discrete alarms
   1: '1000 Betriebsfehler liegt vor / 1000 Operation Error / 1000 Erreur de fonctionnement', class Errors, trigger "WP231PR_DB_s_IO_DATA_OPERATION_ERRORS" bit 0
   2: 'Betriebsfehler Byte 1 Bit 1 / Operation Error Byte 1 Bit 1 / 1101 Court circuit pesons', class Errors, trigger "WP231PR_DB_s_IO_DATA_OPERATION_ERRORS" bit 1
   3: '1104 ADC Sense-Spannung zu gering / 1104 ADC sense voltage too low / 1104 Tension capteurs CAN trop basse', class Errors, trigger "WP231PR_DB_s_IO_DATA_OPERATION_ERRORS" bit 2
   4: 'Betriebsfehler Byte 1 Bit 3 / Operation Error Byte 1 Bit 1 / 1101 Court circuit pesons', class Errors, trigger "WP231PR_DB_s_IO_DATA_OPERATION_ERRORS" bit 3
   5: '1105 ADC Ausserhalb zulässigem Digit-Bereich (positiv) / 1105 ADC out of range (positive) / 1105 CAN hors plage de mesure (max)', class Errors, trigger "WP231PR_DB_s_IO_DATA_OPERATION_ERRORS" bit 4
   6: '1106 ADC Ausserhalb zulässigem Digit-Bereich (negativ) / 1106 ADC out of range (negative) / 1106 CAN hors plage de mesure (min)', class Errors, trigger "WP231PR_DB_s_IO_DATA_OPERATION_ERRORS" bit 5
   7: '1002 RAM-Fehler / 1002 RAM error / 1002 Erreur RAM', class Errors, trigger "WP231PR_DB_s_IO_DATA_OPERATION_ERRORS" bit 6
   8: '1102 ADC Fehler / 1102 ADC error / 1102 Erreur CAN', class Errors, trigger "WP231PR_DB_s_IO_DATA_OPERATION_ERRORS" bit 7
   9: '1005 Prozessalarm verloren / 1005 Processalarm lost / 1005 Perte des messages processus', class Errors, trigger "WP231PR_DB_s_IO_DATA_OPERATION_ERRORS" bit 8
   10: '1003 Checksummenfehler Daten / 1003 Checksum error data / 1003 Erreur données checksum', class Errors, trigger "WP231PR_DB_s_IO_DATA_OPERATION_ERRORS" bit 9
   11: '1107 Eichfähige HMI-Anzeige ist ausgefallen / 1107 Legal-for-trade display disturbed / 1107 Perte de l'affichage légal sur le pupitre HMI', class Errors, trigger "WP231PR_DB_s_IO_DATA_OPERATION_ERRORS" bit 10
   12: '1004 Checksummenfehler Programm / 1004 Checksum error program / 1004 Erreur données checksum du programme', class Errors, trigger "WP231PR_DB_s_IO_DATA_OPERATION_ERRORS" bit 11
   13: '1006 Fehler Logbuch / 1006 Error log-book / 1006 Erreur sur le cahier des rapports', class Errors, trigger "WP231PR_DB_s_IO_DATA_OPERATION_ERRORS" bit 12
   14: '1001 Reset nach Fehler (Watchdog Error) / 1001 Restart after failure (watchdog error) / 1001 Reset après erreur (Watchdog)', class Errors, trigger "WP231PR_DB_s_IO_DATA_OPERATION_ERRORS" bit 13
   15: '1007 Falsche Applikations-ID / 1007 Wrong application ID / 1007 Erreur ID de l'application', class Errors, trigger "WP231PR_DB_s_IO_DATA_OPERATION_ERRORS" bit 14
   16: 'Betriebsfehlerbyte 2 Bit 7 / Operation Error Byte 2 Bit 7 / Erreur fonctionnement octet 2 bit 7', class Errors, trigger "WP231PR_DB_s_IO_DATA_OPERATION_ERRORS" bit 15
   17: '2000 Technologiefehler / 2000 Technological error / 2000 Erreur technologique', class Errors, trigger "WP231PR_DB_s_IO_DATA_TECHNOLOGICAL_ERRORS" bit 0
   18: '2001 Timeout Tarieren oder Nullstellen / 2001 Timeout tare or zero setting / 2001 Timeout tarage ou RAZ (temps d'attente dépassé)', class Errors, trigger "WP231PR_DB_s_IO_DATA_TECHNOLOGICAL_ERRORS" bit 1
   19: '2002 Trace überlastet / 2002 Trace overloaded / 2002 Mémoire trace pleine', class Errors, trigger "WP231PR_DB_s_IO_DATA_TECHNOLOGICAL_ERRORS" bit 2
   20: '2003 Einschaltnullsetzen nicht möglich / 2003 Initial Zeroing not possible / 2003 RAZ à la mise sous tension impossible', class Errors, trigger "WP231PR_DB_s_IO_DATA_TECHNOLOGICAL_ERRORS" bit 3
   21: 'Technologiefehlerbyte 1 Bit 4 / Technological error Byte 1 Bit 4 / Erreur technologique octet 1 bit 4', class Errors, trigger "WP231PR_DB_s_IO_DATA_TECHNOLOGICAL_ERRORS" bit 4
   22: 'Technologiefehlerbyte 1 Bit 5 / Technological error Byte 1 Bit 5 / Erreur technologique octet 1 bit 5', class Errors, trigger "WP231PR_DB_s_IO_DATA_TECHNOLOGICAL_ERRORS" bit 5
   23: 'Technologiefehlerbyte 1 Bit 6 / Technological error Byte 1 Bit 6 / Erreur technologique octet 1 bit 6', class Errors, trigger "WP231PR_DB_s_IO_DATA_TECHNOLOGICAL_ERRORS" bit 6
   24: 'Technologiefehlerbyte 1 Bit 7 / Technological error Byte 1 Bit 7 / Erreur technologique octet 1 bit 7', class Errors, trigger "WP231PR_DB_s_IO_DATA_TECHNOLOGICAL_ERRORS" bit 7
   25: 'Technologiefehlerbyte 1 Bit 7 / Technological error Byte 2 Bit 0 / Erreur technologique octet 2 bit 0', class Errors, trigger "WP231PR_DB_s_IO_DATA_TECHNOLOGICAL_ERRORS" bit 8
   26: 'Technologiefehlerbyte 2 Bit 1 / Technological error Byte 2 Bit 1 / Erreur technologique octet 2 bit 1', class Errors, trigger "WP231PR_DB_s_IO_DATA_TECHNOLOGICAL_ERRORS" bit 9
   27: 'Technologiefehlerbyte 2 Bit 2 / Technological error Byte 2 Bit 2 / Erreur technologique octet 2 bit 2', class Errors, trigger "WP231PR_DB_s_IO_DATA_TECHNOLOGICAL_ERRORS" bit 10
   28: 'Technologiefehlerbyte 2 Bit 3 / Technological error Byte 2 Bit 3 / Erreur technologique octet 2 bit 3', class Errors, trigger "WP231PR_DB_s_IO_DATA_TECHNOLOGICAL_ERRORS" bit 11
   29: 'Technologiefehlerbyte 2 Bit 4 / Technological error Byte 2 Bit 4 / Erreur technologique octet 2 bit 4', class Errors, trigger "WP231PR_DB_s_IO_DATA_TECHNOLOGICAL_ERRORS" bit 12
   30: 'Technologiefehlerbyte 2 Bit 5 / Technological error Byte 2 Bit 5 / Erreur technologique octet 2 bit 5', class Errors, trigger "WP231PR_DB_s_IO_DATA_TECHNOLOGICAL_ERRORS" bit 13
   31: 'Technologiefehlerbyte 2 Bit 6 / Technological error Byte 2 Bit 6 / Erreur technologique octet 2 bit 6', class Errors, trigger "WP231PR_DB_s_IO_DATA_TECHNOLOGICAL_ERRORS" bit 14
   32: 'Technologiefehlerbyte 2 Bit 7 / Technological error Byte 2 Bit 7 / Erreur technologique octet 2 bit 7', class Errors, trigger "WP231PR_DB_s_IO_DATA_TECHNOLOGICAL_ERRORS" bit 15
   33: '5000 Daten- oder Bedienfehler / 5000 Data or command error / 5000 Erreur données ou utilisateur', class Errors, trigger "WP231PR_DB_s_IO_DATA_DATA_CMD_ERROR_1" bit 0
   34: '5001 Befehlscode oder Datensatz nicht bekannt / 5001 Data record or command unknown / 5001 Ordre ou numéro de DR inconnu', class Errors, trigger "WP231PR_DB_s_IO_DATA_DATA_CMD_ERROR_1" bit 1
   35: '5002 Befehl oder Datenänderung nicht erlaubt, da Schreibschutz aktiv / 5002 Command or Data modification not allowed / 5002 Ordre ou modification des paramètres interdit parce que la protection en écriture est activée', class Errors, trigger "WP231PR_DB_s_IO_DATA_DATA_CMD_ERROR_1" bit 2
   36: '5003 Verlassen des Servicebetriebs unzulässig, da Justage nicht abgeschlossen / 5003 Service Mode can't be switched off, as calibration was not completed / 5003 Impossible de quitter le mode service parce que l'étalonnage n'est pas terminé', class Errors, trigger "WP231PR_DB_s_IO_DATA_DATA_CMD_ERROR_1" bit 3
   37: '5004 Befehl oder Datenübertragung nur im Servicebetrieb möglich / 5004 Command or data transfer only permitted in service mode / 5004 Ordre ou transmission de données uniquement possible en mode service', class Errors, trigger "WP231PR_DB_s_IO_DATA_DATA_CMD_ERROR_1" bit 4
   38: '5005 Befehl oder Datenübertragung im Servicebetrieb nicht möglich, da Servicebetrieb aktiv / 5005 Command or data transfer not permitted in service mode / 5005 Ordre ou transmission de données impossible parce que le mode service est activé', class Errors, trigger "WP231PR_DB_s_IO_DATA_DATA_CMD_ERROR_1" bit 5
   39: '5006 Befehl oder Datenübertragung nicht möglich da BUSY / 5006 Command or data transfer not possible while BUSY / 5006 Ordre ou transmission de données impossible parce que la CPU est en mode stop ou erreur', class Errors, trigger "WP231PR_DB_s_IO_DATA_DATA_CMD_ERROR_1" bit 6
   40: '5007 Befehl oder Datenübertragung nicht möglich da Modul gestört oder CPU in Stop / 5007 Command or data transfer not possible because of error or CPU stop / 5007 Ordre ou transmission de données impossible parce que le module est en mode BUSY', class Errors, trigger "WP231PR_DB_s_IO_DATA_DATA_CMD_ERROR_1" bit 7
   41: 'Daten-Bedienfehler Byte 2 Bit 0 / Data Command Error Byte 2 Bit 0 / Erreur de données/d'utilisation octet 2 bit 0', class Errors, trigger "WP231PR_DB_s_IO_DATA_DATA_CMD_ERROR_1" bit 8
   42: '5103 Befehl nicht möglich, da Eichanzeige fehlt oder nicht sichtbar / 5103 Command not possible - SecureDisplay is missing or hidden / 5103 Ordre impossible parce que l'afficheur légal manque ou n'est pas disponible', class Errors, trigger "WP231PR_DB_s_IO_DATA_DATA_CMD_ERROR_1" bit 9
   43: '5101 Befehle in diesem Zustand nicht möglich / 5101 Command in this state not possible / 5101 Ordre impossible dans cet état', class Errors, trigger "WP231PR_DB_s_IO_DATA_DATA_CMD_ERROR_1" bit 10
   44: '5102 Befehl nicht möglich, da kein Stillstand vorliegt / 5102 Command not possible - No Standstill / 5102 Ordre impossible parce que l'état stable n'est pas atteint', class Errors, trigger "WP231PR_DB_s_IO_DATA_DATA_CMD_ERROR_1" bit 11
   45: '5104 Befehl nicht möglich, da Bereich überschritten / 5104 Command not possible - Limit exceeded / 5104 Ordre impossible parce que la plage de mesure est dépassée', class Errors, trigger "WP231PR_DB_s_IO_DATA_DATA_CMD_ERROR_1" bit 12
   46: '5105 Wägezellenparameter nicht plausibel / 5105 Load cell parameter not plausible / 5105 Les paramètres pesons ne sont pas plausibles', class Errors, trigger "WP231PR_DB_s_IO_DATA_DATA_CMD_ERROR_1" bit 13
   47: 'Daten-Bedienfehler Byte 2 Bit 0 / Data Command Error Byte 2 Bit 6 / Erreur de données/d'utilisation octet 2 bit 6', class Errors, trigger "WP231PR_DB_s_IO_DATA_DATA_CMD_ERROR_1" bit 14
   48: '5107 Kennlinienverschiebung nicht möglich / 5107 Calibration charcteristic shift not possible / 5107 Translation de la courbe caractéristique impossible', class Errors, trigger "WP231PR_DB_s_IO_DATA_DATA_CMD_ERROR_1" bit 15
   49: '5109 Protokollierung nicht möglich, da seit letzter Protokollierung keine Messwertänderung stattgefunden hat / 5109 Logging not possible, as the weight value did not change since the last logging / 5109 Mémorisation du rapport impossible parceque le poids n'a pas changé depuis le dernier rapport', class Errors, trigger "WP231PR_DB_s_IO_DATA_DATA_CMD_ERROR_2" bit 0
   50: 'Daten-Bedienfehler Byte 2 Bit 0 / Data Command Error Byte 3 Bit 1 / Erreur de données/d'utilisation octet 3 bit 1', class Errors, trigger "WP231PR_DB_s_IO_DATA_DATA_CMD_ERROR_2" bit 1
   51: 'Daten-Bedienfehler Byte 2 Bit 0 / Data Command Error Byte 3 Bit 2 / Erreur de données/d'utilisation octet 3 bit 2', class Errors, trigger "WP231PR_DB_s_IO_DATA_DATA_CMD_ERROR_2" bit 2
   52: 'Daten-Bedienfehler Byte 2 Bit 0 / Data Command Error Byte 3 Bit 3 / Erreur de données/d'utilisation octet 3 bit 3', class Errors, trigger "WP231PR_DB_s_IO_DATA_DATA_CMD_ERROR_2" bit 3
   53: 'Daten-Bedienfehler Byte 2 Bit 0 / Data Command Error Byte 3 Bit 4 / Erreur de données/d'utilisation octet 3 bit 4', class Errors, trigger "WP231PR_DB_s_IO_DATA_DATA_CMD_ERROR_2" bit 4
   54: '5199 Fehler bei Befehl an DE / 5199 Error caused by command on DI / 5199 Erreur d'ordre entré par une entrée TOR', class Errors, trigger "WP231PR_DB_s_IO_DATA_DATA_CMD_ERROR_2" bit 5
   55: 'Daten-Bedienfehler Byte 2 Bit 0 / Erreur de données/d'utilisation octet 3 bit 6', class Errors, trigger "WP231PR_DB_s_IO_DATA_DATA_CMD_ERROR_2" bit 6
   56: 'Daten-Bedienfehler Byte 2 Bit 0 / Data Command Error Byte 3 Bit 7 / Erreur de données/d'utilisation octet 3 bit 7', class Errors, trigger "WP231PR_DB_s_IO_DATA_DATA_CMD_ERROR_2" bit 7
   57: 'Daten-Bedienfehler Byte 4 Bit 0 / Data Command Error Byte 4 Bit 0 / Erreur de données/d'utilisation octet 4 bit 0', class Errors, trigger "WP231PR_DB_s_IO_DATA_DATA_CMD_ERROR_2" bit 8
   58: 'Daten-Bedienfehler Byte 4 Bit 1 / Data Command Error Byte 4 Bit 1 / Erreur de données/d'utilisation octet 4 bit 1', class Errors, trigger "WP231PR_DB_s_IO_DATA_DATA_CMD_ERROR_2" bit 9
   59: 'Daten-Bedienfehler Byte 4 Bit 2 / Data Command Error Byte 4 Bit 2 / Erreur de données/d'utilisation octet 4 bit 2', class Errors, trigger "WP231PR_DB_s_IO_DATA_DATA_CMD_ERROR_2" bit 10
   60: '6002 Protokollieren nicht möglich, da Gewicht unzulässig / 6002 Logging not possible - Weight not plausible / 6002 Impossible d'écrire le rapport, le poids est hors tolérances', class Errors, trigger "WP231PR_DB_s_IO_DATA_DATA_CMD_ERROR_2" bit 11
   61: '5108 Logbuch-ID nicht vorhanden / 5108 Log ID not existing / 5108 Carnet de rapport n'existe pas', class Errors, trigger "WP231PR_DB_s_IO_DATA_DATA_CMD_ERROR_2" bit 12
   62: 'Daten-Bedienfehler Byte 4 Bit 2 / Data Command Error Byte 4 Bit 5 / Erreur de données/d'utilisation octet 4 bit 5', class Errors, trigger "WP231PR_DB_s_IO_DATA_DATA_CMD_ERROR_2" bit 13
   63: 'Daten-Bedienfehler Byte 4 Bit 2 / Data Command Error Byte 4 Bit 6 / Erreur de données/d'utilisation octet 4 bit 6', class Errors, trigger "WP231PR_DB_s_IO_DATA_DATA_CMD_ERROR_2" bit 14
   64: 'Daten-Bedienfehler Byte 4 Bit 2 / Data Command Error Byte 4 Bit 7 / Erreur de données/d'utilisation octet 4 bit 7', class Errors, trigger "WP231PR_DB_s_IO_DATA_DATA_CMD_ERROR_2" bit 15
   65: '7000 Zulässiger Zahlenbereich verlassen / 7000 Counting range exceeded / 7000 Hors plage numérique', class Errors, trigger "WP231PR_DB_s_IO_DATA_DATA_CMD_ERROR_3" bit 0
   66: 'Daten-Bedienfehler Byte 5 Bit 1 / Data Command Error Byte 5 Bit 1 / Erreur de données/d'utilisation octet 5 bit 1', class Errors, trigger "WP231PR_DB_s_IO_DATA_DATA_CMD_ERROR_3" bit 1
   67: '7001 Vorschriftencode nicht bekannt / 7001 Restriction code unknown / 7001 Code métrologique inconnu', class Errors, trigger "WP231PR_DB_s_IO_DATA_DATA_CMD_ERROR_3" bit 2
   68: 'Daten-Bedienfehler Byte 5 Bit 3 / Data Command Error Byte 5 Bit 3 / Erreur de données/d'utilisation octet 5 bit 1', class Errors, trigger "WP231PR_DB_s_IO_DATA_DATA_CMD_ERROR_3" bit 3
   69: '7003 Vorgabe Datum/Uhrzeit nicht plausibel / 7003 Date / Time parameter not plausible / 7003 Consigne de date/heure pas plausible', class Errors, trigger "WP231PR_DB_s_IO_DATA_DATA_CMD_ERROR_3" bit 4
   70: '7004 Zuordnung DQ/DI nicht plausibel / 7004 Assignment of digital input or output not plausible / 7004 Affectation des entrées/sorties TOR erronée', class Errors, trigger "WP231PR_DB_s_IO_DATA_DATA_CMD_ERROR_3" bit 5
   71: 'Daten-Bedienfehler Byte 5 Bit 6 / Data- / Command Error Byte 5 Bit 6 / 7006 Ordre réservé pour banc de test usine', class Errors, trigger "WP231PR_DB_s_IO_DATA_DATA_CMD_ERROR_3" bit 6
   72: '7007 Die Justagegewichte bzw. Justagedigits sind nicht plausibel / 7007 Calibrationweights / Calibrationdigits not plausible / 7007 Les poids étalons ou les digits d'étalonnage ne sont pas plausibles', class Errors, trigger "WP231PR_DB_s_IO_DATA_DATA_CMD_ERROR_3" bit 7
   73: '7008 Nullstell- / Nullsetz- oder Taraparameter nicht plausibel / 7008 Zero- / Tare weights not plausible / 7008 Les valeur de RAZ ne sont pas plausibles', class Errors, trigger "WP231PR_DB_s_IO_DATA_DATA_CMD_ERROR_3" bit 8
   74: '7009 Stillstandsbereich / Stillstandswartezeit nicht plausibel / 7009 Standstillrange / Standstilltime not plausible / 7009 Les valeurs de tempo ou de poids pour l'état stable ne sont pas plausibles', class Errors, trigger "WP231PR_DB_s_IO_DATA_DATA_CMD_ERROR_3" bit 9
   75: '7010 Ziffernschritt / Rundung nicht plausibel / 7010 Numeral step / rounding not plausible / 7010 Echelon ou arrondit ne sont pas plausibles', class Errors, trigger "WP231PR_DB_s_IO_DATA_DATA_CMD_ERROR_3" bit 10
   76: '7011 Filterparameter nicht plausibel / 7011 Filter parameter not plausible / 7011 Les paramètres des filtres ne sont pas plausibles', class Errors, trigger "WP231PR_DB_s_IO_DATA_DATA_CMD_ERROR_3" bit 11
   77: '7013 Schnittstellenparameter SecureDisplay nicht plausibel / 7013 Interface settings for legal display not plausible / 7013 Les paramètres de SecureDisplay ne sont pas plausibles', class Errors, trigger "WP231PR_DB_s_IO_DATA_DATA_CMD_ERROR_3" bit 12
   78: '7014 Zeitvorgabe nicht plausibel / 7014 Time value not plausible / 7014 de données/d'utilisation octet 6 bit 5', class Errors, trigger "WP231PR_DB_s_IO_DATA_DATA_CMD_ERROR_3" bit 13
   79: 'Daten-Bedienfehler Byte 6 Bit 6 / Data- / Command Error Byte 6 Bit 6 / Erreur de données/d'utilisation octet 6 bit 6', class Errors, trigger "WP231PR_DB_s_IO_DATA_DATA_CMD_ERROR_3" bit 14
   80: '7016 Parametrierung des Analogausgangs ist nicht plausibel / 7016 Analog output parameter not plausible / 7016 Le paramétrage de la sortie analogique n'est pas plausible', class Errors, trigger "WP231PR_DB_s_IO_DATA_DATA_CMD_ERROR_3" bit 15
   81: '7017 MAC Adresse kann nicht geändert werden / 7017 MAC address can not be changed / 7017 Impossible de changer l'adresse MAC', class Errors, trigger "WP231PR_DB_s_IO_DATA_DATA_CMD_ERROR_4" bit 0
   82: '7018 Fehler in IP-Maske / 7018 Error in IP mask / 7018 Erreur dans la vue IP', class Errors, trigger "WP231PR_DB_s_IO_DATA_DATA_CMD_ERROR_4" bit 1
   83: '7019 RS485 Parameter nicht plausibel / 7019 RS485 parameter not plausible / 7019 Les paramètres RS485 ne sont pas plausibles', class Errors, trigger "WP231PR_DB_s_IO_DATA_DATA_CMD_ERROR_4" bit 2
   84: 'Daten-Bedienfehler Byte 7 Bit 4 / Data- / Command Error Byte 7 Bit 3 / Erreur de données/d'utilisation octet 7 bit 3', class Errors, trigger "WP231PR_DB_s_IO_DATA_DATA_CMD_ERROR_4" bit 3
   85: 'Daten-Bedienfehler Byte 7 Bit 5 / Data- / Command Error Byte 7 Bit 4 / Erreur de données/d'utilisation octet 7 bit 4', class Errors, trigger "WP231PR_DB_s_IO_DATA_DATA_CMD_ERROR_4" bit 4
   86: 'Daten-Bedienfehler Byte 7 Bit 6 / Data- / Command Error Byte 7 Bit 5 / Erreur de données/d'utilisation octet 7 bit 5', class Errors, trigger "WP231PR_DB_s_IO_DATA_DATA_CMD_ERROR_4" bit 5
   87: 'Daten-Bedienfehler Byte 7 Bit 7 / Data- / Command Error Byte 7 Bit 6 / Erreur de données/d'utilisation octet 7 bit 6', class Errors, trigger "WP231PR_DB_s_IO_DATA_DATA_CMD_ERROR_4" bit 6
   88: 'Daten-Bedienfehler Byte 8 Bit 0 / Data- / Command Error Byte 7 Bit 7 / Erreur de données/d'utilisation octet 7 bit 7', class Errors, trigger "WP231PR_DB_s_IO_DATA_DATA_CMD_ERROR_4" bit 7
   89: 'Daten-Bedienfehler Byte 8 Bit 1 / Data- / Command Error Byte 8 Bit 0 / Erreur de données/d'utilisation octet 8 bit 0', class Errors, trigger "WP231PR_DB_s_IO_DATA_DATA_CMD_ERROR_4" bit 8
   90: 'Daten-Bedienfehler Byte 8 Bit 2 / Data- / Command Error Byte 8 Bit 1 / Erreur de données/d'utilisation octet 8 bit 1', class Errors, trigger "WP231PR_DB_s_IO_DATA_DATA_CMD_ERROR_4" bit 9
   91: 'Daten-Bedienfehler Byte 8 Bit 3 / Data- / Command Error Byte 8 Bit 2 / Erreur de données/d'utilisation octet 8 bit 2', class Errors, trigger "WP231PR_DB_s_IO_DATA_DATA_CMD_ERROR_4" bit 10
   92: 'Daten-Bedienfehler Byte 8 Bit 4 / Data- / Command Error Byte 8 Bit 3 / Erreur de données/d'utilisation octet 8 bit 3', class Errors, trigger "WP231PR_DB_s_IO_DATA_DATA_CMD_ERROR_4" bit 11
   93: 'Daten-Bedienfehler Byte 8 Bit 5 / Data- / Command Error Byte 8 Bit 4 / Erreur de données/d'utilisation octet 8 bit 4', class Errors, trigger "WP231PR_DB_s_IO_DATA_DATA_CMD_ERROR_4" bit 12
   94: 'Daten-Bedienfehler Byte 8 Bit 6 / Data- / Command Error Byte 8 Bit 5 / Erreur de données/d'utilisation octet 8 bit 5', class Errors, trigger "WP231PR_DB_s_IO_DATA_DATA_CMD_ERROR_4" bit 13
   95: 'Daten-Bedienfehler Byte 8 Bit 6 / Data- / Command Error Byte 8 Bit 6 / Erreur de données/d'utilisation octet 8 bit 6', class Errors, trigger "WP231PR_DB_s_IO_DATA_DATA_CMD_ERROR_4" bit 14
   96: 'Daten-Bedienfehler Byte 8 Bit 6 / Data- / Command Error Byte 8 Bit 6 / Erreur de données/d'utilisation octet 8 bit 7', class Errors, trigger "WP231PR_DB_s_IO_DATA_DATA_CMD_ERROR_4" bit 15

text list "013010_RS485_BAUD_RATE": 2 '9600 Bit/s'; 3 '19200 Bit/s'; 4 '38400 Bit/s'; 5 '57600 Bit/s'; 6 '115000 Bit/s'

text list "013012_RS485_PARITY": 0 'gerade / even / pair'; 1 'ungerade / odd / impair'

text list "013012_RS485_DATA_BITS": 0 '7 Datenbits / 7 Data Bits'; 1 '8 Datenbits / 8 Data Bits'

text list "013008_RS485_PROTOCOL": 0 'Kein Gerät / No Device / Aucun appareil'; 1 'Modbus RTU'; 2 'Siebert-Display S102'

text list "013016_DECIMAL_POINTS_REMOTE_DISPLAY": 0 'Keine Nachkommastelle / No decimal point / Pas de point décimal / No decimal points'; 1 'Eine Nachkommastelle / 1 decimal point / 1 décimale après la virgule / One decimal point'; 2 'Zwei Nachkommastellen / Two decimal points / Deux décimales'; 3 'Drei Nachkommastellen / 3 decimal points / 3 décimales après la virgule / Three decimal points'; 4 'Vier Nachkommastellen / Four decimal points / Quatre décimales'

text list "013012_RS485_STOP_BITS": 0 '1 Stop Bit'; 1 '2 Stop Bits'

text list "014008_SELECTION_PROC_VAL_1_S7": 0 'Kein Element selektiert / No element selected / Aucun élément sélectionné'; 1 'Brutto Prozesswert (F1) / Gross process weight (F1) / Poids brut processus (F1)'; 2 'Netto Prozesswert (F1) / Net process weight (F1) / Net processus (F1)'; 3 'Tara Prozesswert / Tare process weight / Poids tare (processus)'; 4 'Brutto/Netto Gewicht (OIML) / Gross/Net weight (legal) / Poids brut/net processus (OIML)'; 5 'B/N Gewicht x 10 / Gross/Net weight x10 / Poids brut / Net x 10'; 6 'Tara Gewicht (OIML) / Tare weight (legal) / Tare poids mode OIML'; 7 'Brutto Prozesswert (F2) / Gross process weight (F2) / Poids brut processus (F2)'; 8 'Netto Prozesswert (F2) / Net process weight (F2) / Net processus (F2)'; 9 'Ungefilterter Digitwert / Digits unfiltered / Valeur CAN non filtrée'; 10 'Gefilterter Digitwert (F1) / Digits filtered (F1) / Valeur CAN filtrée (F1)'; 11 'Gefilterter Digitwert (F2) / Digits filtered (F2) / Valeur CAN filtrée (F2)'; 12 'Refresh Counter / Rafraichissement compteur'; 13 'Status AA-DA-DE / Status AO-DO-DI / Etat E/S TOR'

text list "014010_SELECTION_PROC_VAL_2_S7": 0 'Kein Element selektiert / No element selected / Aucun élément sélectionné'; 1 'Brutto Prozesswert (F1) / Gross process weight / Poids brut processus (F1)'; 2 'Netto Prozesswert (F1) / Net process weight / Net processus (F1)'; 3 'Tara Prozesswert / Tare process weight / Poids tare (processus)'; 4 'Brutto/Netto Gewicht (OIML) / Gross/Net weight (legal) / Poids brut/net processus (OIML)'; 5 'B/N Gewicht x 10 / Gross/Net weight x10 / Poids brut / Net x 10'; 6 'Tara Gewicht (OIML) / Tare weight (legal) / Tare poids mode OIML'; 7 'Brutto Prozesswert (F2) / Gross process weight (F2) / Poids brut processus (F2)'; 8 'Netto Prozesswert (F2) / Net process weight (F2) / Net processus (F2)'; 9 'Ungefilterter Digitwert / Digits unfiltered / Valeur CAN non filtrée'; 10 'Gefilterter Digitwert (F1) / Digits filtered (F1) / Valeur CAN filtrée (F1)'; 11 'Gefilterter Digitwert (F2) / Digits filtered (F2) / Valeur CAN filtrée (F2)'; 12 'Refresh Counter / Rafraichissement compteur'; 13 'Status AA-DA-DE / Status AO-DO-DI / Etat E/S TOR'

text list "003030_LETTER_FOR_GROSS_WEIGHT": 66 'B für Brutto / B for Gross / B pour Brut'; 71 'G für Brutto / G for Gross / G pour Brut'

text list "007020_ASSIGNMENT_DIGITAL_OUTPUT": 0 '1/4d Null / 1/4 d Zero / 1/4 d zéro'; 1 'Max 9e / max 9e'; 2 'Tariert / tared / taré'; 3 'Hand-Tara gesetzt (pT) / Preset Tara active (pT) / Tare manuelle (pT)'; 6 'Status Stillstand / Stand Still / Etat stable'; 8 'Leer / Grenzwert 3 / Empty / Limit 3 / Vide / Limite 3'; 9 'Grenzwert 1 / Limit 1 / Limite 1'; 10 'Grenzwert 2 / Limit 2 / Limite 2'; 11 'Min unterschritten / Below Min / Sous le minimum'; 22 'Trace aktiv / Trace active'; 23 'Bedienfehler durch digit. Eingang / Comand error by Digit. Input / Erreur commande par entrée TOR'; 24 'Waage justiert / Scale calibrated / Balance étalonnée'; 25 'Servicebetrieb / Service Mode / Mode service'; 26 'Simulationsbetrieb / Simulation mode / Mode simulation'; 27 'Schreibschutz / Write Protection / Protection écriture'; 28 'Analogausgang gestört / Analog output error / Erreur sortie analogique'; 30 'Anlauf / Start up / Démarrage'; 31 'Störung / Error / Erreur'; 33 'Test / Steuern Ausgang / Test / Force Output / Test sortie TOR'; 34 'Test / Steuern über S7 Schnittstelle / Test / Force by S7 interface / Test par interface API S7'; 255 'deaktiviert / disabled / Sortie désactivée'; 109 'Grenzwert 1 (invertiert) / Limit 1 (inverted) / Limite 1 (inversé)'; 110 'Grenzwert 2 (invertiert) / Limit 2 (inverted) / Limite 2 (inversé)'; 108 'Leer / Grenzwert 3 (invertiert) / Empty / Limit 3 (inverted) / Vide / Limite 3 (inversé)'; 128 'Analogausgang gestört (invertiert) / Analog output error (inverted) / Erreur sortie analogique (inversé)'; 131 'Störung (invertiert) / Error (inverted) / Erreur (inversé)'

text list "007026_DIGIT_STATUS_BY_ERROR_STOP": 0 'Alle "AUS" / All "FALSE" / Tous "on"'; 1 'Funktion erhalten / Obtain functionality / Garder la fonction'; 2 'Definierte Ersatzwerte / Defined Value / Valeur de remplacement'; 3 'Alle "EIN" / All "TRUE" / Tous "off"'

text list "003072_FALSE_TRUE": 0 'AUS / FALSE / Arrêt'; 1 'EIN / TRUE / Marche'

text list "FORCE_DIGITAL_IO": 0 'STEUERN "AUS" / Force "OFF" / Contrôle "off"'; 1 'STEUERN "EIN" / Force "ON" / Contrôle "on"'

text list "007030_RANGE_ANALOG_OUTPUT": 0 '0...20 mA'; 1 '4...20 mA'

text list "DAY_OF_WEEK": 1 'Sonntag / Sunday / Dimanche'; 2 'Montag / Monday / Lundi'; 3 'Dienstag / Tuesday / Mardi'; 4 'Mittwoch / Wednesday / Mercredi'; 5 'Donnerstag / Thursday / Jeudi'; 6 'Freitag / Friday / Vendredi'; 7 'Samstag / Saturday / Samedi'

text list "007032_SOURCE_ANALOG_OUTPUT": 0 'Brutto/Netto Gewicht / Gross/Net Weight / Poids brut/net processus'; 1 'Bruttogewicht / Gross Weight / Poids brut'; 2 'Nettogewicht / Net Weight / Poids net'; 3 'Test / Steuern Analogausgang / Test / Force Output / Test / sortie analogique'; 4 'Steuern über S7 Schnittstelle / Test / Force by S7 interface / Test par interface API S7'

text list "006008_BASIS_FOR_LIMITS_1_2": 0 'Bruttogewicht (% von Max. Wägebereich) / Gross Weight (% of max. weight) / Poids brut (% du poids max.)'; 1 'Nettogewicht (% von Max. Wägebereich) / Net Weight (% of max. weight) / Poids net (% du poids max.)'; 2 'Bruttogewicht (Absolutwert) / Gross Weight (absolut value) / Poids brut (valeur absolue)'; 3 'Nettogewicht (Absolutwert) / Net Weight (absolut value) / Poids net (valeur absolue)'

text list "003112_ORDER_NO_LOW_PASS_FILTER": 2 '2'; 4 '4'; 6 '6'; 8 '8'; 10 '10'

text list "003072_NO_YES": 0 'nein / no / non'; 1 'ja / yes / oui'

text list "003074_ROUNDING_PROCESS_VAL": 1 'Rundung auf 1 Nachkommastelle / Rounding after 1 decimal point / Arrondi à 1 décimale / One decimal point'; 2 'Rundung auf 2 Nachkommastellen / Rounding after 2 decimal points / Arrondi à 2 décimales / One decimal point'; 3 'Rundung auf 3 Nachkommastellen / Rounding after 3 decimal points / Arrondi à 3 décimales / One decimal point'; 4 'Rundung auf 4 Nachkommastellen / Rounding after 4 decimal points / Arrondi à 4 décimales / One decimal point'; 5 'Rundung auf 5 Nachkommastellen / Rounding after 5 decimal points / Arrondi à 5 décimales / One decimal point'; 6 'Rundung auf 6 Nachkommastellen / Rounding after 6 decimal points / Arrondi à 6 décimales / One decimal point'; 0 'Keine Rundung / No Rounding / Pas d'arrondit'

text list "007034_ANALOG_STATUS_BY_ERROR_STOP": 0 'Min. (0mA) / min (0mA)'; 1 'Funktion erhalten / Obtain functionality / Garder la fonction'; 2 'Definierter Ersatzwert / Defined Value / Valeur de remplacement'; 3 'Max. (24mA)'

text list "007048_TRACE_RATE": 1 '10 ms'; 10 '100 ms'; 100 '1 s'; 1000 '10 s'

text list "007050_TRACE_MEMORY_TYPE": 0 'Speicher überschreiben (Ringspeicher) / Memory overwrite (Ringbuffer) / Réécriture de la mémoire'; 1 'Stop bei vollem Speicher / Stop when Memory is full / Arrêt quand mémoire pleine'

text list "007008_ASSIGNMENT_DIGITAL_INPUT": 0 'deaktiviert / disabled / Inactif'; 1 'Servicebetrieb ein (1) / Service Mode On (1) / Mode service (1)'; 2 'Servicebetrieb aus (2) / Service Mode Off (2) / Arrêt mode service (2)'; 3 'Simulation ein (3) / Weight Simulation on (3) / Simulation poids (3)'; 4 'Simulation aus (4) / Weight Simulation off (4) / Arrêt simulation (4)'; 11 'Werkseinstellung laden (11) / Load Factory Settings (11) / Configuration usine (11)'; 31 'Alle Parameter wiederherstellen (31) / Restore all weighing parameters (31) / Charger param sauvegarde (31)'; 51 'Alle Parameter speichern (51) / Create Recovery Parameter (51) / Créer param sauvegarde (51)'; 60 'Justagepunkt 0 gültig (60) / Set Calibration Point 0 (60) / Poids étalon 0 (60)'; 61 'Justagepunkt 1 gültig (61) / Set Calibration Point 1 (61) / Poids étalon 1 (61)'; 62 'Justagepunkt 2 gültig (62) / Set Calibration Point 2 (62) / Poids étalon 2 (62)'; 81 'Kennlinienverschiebung (81) / Shift Characteristics (81) / Déplace courbe caract. (81)'; 82 'Automatische Justage (82) / Automatic Calibration (82) / Etalonnage automatique (82)'; 1001 'Nullstellen (1001) / Zero (1001) / Zéro (1001)'; 1011 'Tarieren (1011) / Tare (1011)'; 1012 'Tara löschen (1012) / Delete Tare (1012) / Effacement tare (1012)'; 1013 'Taravorgabe 1 gültig (1013) / Set Preset Tare 1 (1013) / Activer Tare 1 (1013)'; 1014 'Taravorgabe 2 gültig (1014) / Set Preset Tare 2 (1014) / Activer Tare 2 (1014)'; 1015 'Taravorgabe 3 gültig (1015) / Set Preset Tare 3 (1015) / Activer Tare 3 (1015)'; 1016 'Taravorgabe S7 gültig (1016) / Set Preset Tare S7 (1016) / Activer Tare S7 (1016)'; 705 'Aktuelles Tara anzeigen (705) / Display Current Tare (705) / Afficher tare actuelle (705)'; 710 'Standardanzeige aktivieren (710) / Display Standard Weight (710) / Activé l'afficheur standard (710)'; 711 'B/N Anzeige aktivieren (711) / Display Gross/Net (711) / Afficher brut/net (711)'; 712 'Netto Anzeige aktivieren (712) / Display Net Weight (712) / Afficher poids net (712)'; 713 'Bruttoanzeige aktivieren (713) / Display Gross Weight (713) / Afficher poids brut (713)'; 714 'Netto Prozessanzeige aktivieren (714) / Display Net Process (714) / Afficher valeur process. net (714)'; 715 'Brutto Prozessanzeige aktivieren (715) / Display Gross Process (715) / Valeur process. brut (715)'; 716 'Brutto Prozessanzeige F2 aktivieren (716) / Display Gross Process F2 (716) / Valeur process. brut filtre F2 (716)'; 801 'Aktuelle Eichvorschrift anzeigen (801) / Display Current Restriction Code (801) / Afficher code métrolo. (801)'; 871 'Aktuelle Seriennummer anzeigen (871) / Display Product Number (871) / Afficher n° cmd. produit (871)'; 875 'Firmwareversion anzeigen (875) / Display Firmware Version (875) / Afficher version firmware (875)'; 876 'Firmwareversion HMI anzeigen (876) / Display HMI-Firmware Version (876) / Afficher Version FW HMI (876)'; 451 'Trace ein (451) / Trace on (451)'; 452 'Trace aus (452) / Trace off (452)'; 453 'Einzeltrace (453) / Trace Single Element (453) / Trace une fois (453)'; 454 'Trace Speicher löschen (454) / Delete Trace Memory (454) / Effacer mémoire trace (454)'

text list "007016_FILTER_DIGITAL_INPUT": 0 '0,2 ms'; 1 '0,2 ms'; 2 '0,4 ms'; 3 '0,8 ms'; 4 '1,6 ms'; 5 '3,2 ms'; 6 '6,4 ms'; 7 '12,8 ms'

text list "RESTRICTION": 0 'Nicht geeichter Betrieb / Non legal for trade / Non soumis à vérification'; 1 'OIML R76 / OIML R-76'

text list "SECURE_DISPLAY_INTERFACE": 0 'kein SecureDisplay / no SecureDisplay / Pas de SecureDisplay'; 1 'An WP231 Port / Via WP231 port / Connexion au WP231'; 2 'An CPU-Port / Via CPU port / Connexion à la CPU'

text list "SHOW_HIDE": 0 'ausblenden / hide / masquer'; 1 'anzeigen / show / afficher'

graphic list "Signal_grey_yellow": 1 'Field Yellow'; 0 'Field Grey'

graphic list "Signal_grey_green": 1 'Field Green'; 0 'Field Grey'

graphic list "Signal_grey_red": 1 'Field Red'; 0 'Field Grey'

screen "2.0_Menu_diagnostic" 800x480, template "Template_1"
   TextField "OBJECT_82" at 0,0 size 220x34; Text '2.0 Diagnose / 2.0 Diagnostics / 2.0 Diagnostic / Diagnostics'
   Button "Go_to_Module_Info" at 416,174 size 350x90; TextOn 'Texte / text'; TextOff '2.5 Trace Start & Stopp / 2.5 Start / Stop Trace / 2.6 Démarrer/arrêter trace / Message List'
      on Press: ActivateScreen("2.5.1_Trace_Start_Stop", 0)
   Button "Exit_to_Main_menue" at 45,390 size 80x80; TextOn 'Texte / text'; TextOff 'Texte / text'; PictureOff "Exit"
      on Press: ActivateScreen("0.0.0_Scale_View_1", 0)
   Button "Go_to_Module_Info_2" at 33,275 size 350x90; TextOn 'Texte / text'; TextOff '2.3 Belastungskurve / 2.3 Load Trend / 2.3 Courbe du poids brut / Message List'
      on Release: SetTag("WP231PR_DB_CMD_B", 2030)
      on Press: ActivateScreen("2.3.0_Load_Trend", 0); SetTag("WP231PR_DB_s_CMD2_i_CMD_CODE", '2003'); SetBit("WP231PR_DB_s_CMD2_bo_CMD_TRIGGER")
   Button "Go_to_Module_Info_1" at 33,174 size 350x90; TextOn 'Texte / text'; TextOff '2.2 Waagenstatus / 2.2 Scale Status / 2.2 Etat de la balance / Message List'
      on Press: ActivateScreen("2.2.1_Scale_Status_1", 0); SetTag("WP231PR_DB_CMD_B", 2034)
   Button "Go_to_Module_Info_3" at 33,73 size 350x90; TextOn 'Texte / text'; TextOff '2.1 Meldungen / 2.1 Messages / Message List'
      on Press: function_ef3f5d25("Messages", -1)
   Button "Go_to_Module_Info_4" at 416,73 size 350x90; TextOn 'Texte / text'; TextOff '2.4 Modulinfo / 2.4 Module Info / 2.4 Infos module / Message List'
      on Press: ActivateScreen("2.4.1_DR9_Modul_info", 0); SetTag("WP231PR_DB_s_CMD2_i_CMD_CODE", '2009'); SetBit("WP231PR_DB_s_CMD2_bo_CMD_TRIGGER")
   Button "Go_to_Module_Info_5" at 416,275 size 350x90; TextOn 'Texte / text'; TextOff '2.6 Erhöhte Auflösung / 2.6 Increased resolution / 2.6 Résolution accrue / Message List'
      on Release: ActivateScreen("0.0.0_Scale_View_1", 0)
      on Press: SetTag("WP231PR_DB_s_CMD2_i_CMD_CODE", 701); SetBit("WP231PR_DB_s_CMD2_bo_CMD_TRIGGER")
   Softkey "[!Invalid!]Softkey_F6" at -140,-147 size 0x0
      on KeyDown: ActivateScreen("0.0.0_Menu_main", 0)

screen "1.5.5_DR17_control_analogue_output" 800x480, template "Template_1"
   TextField "OBJECT_33" at 0,0 size 496x32; Text '1.5.5 Test / Steuern Analog-Ausgang / 1.5.5 Test / Force Analogue Output / 1.5.5 Test & contrôle sortie analogique / Setup 2/3'
   Button "OBJECT_24" at 45,390 size 80x80; TextOn 'Texte / text'; TextOff 'Texte / text'; PictureOff "Exit"
      on Release: ActivateScreen("1.5.0.1_Menu_communication_interfaces_1", 0)
   TextField "OBJECT_10" at 56,301 size 295x32; Text 'Vorgabewert Analogausgang / Test / Force Value / Définition sortie analogique / Display Resolution'
      Visibility <- "WP231PR_DB_DR07_SOURCE_ANA_OUT"
   IOField "OBJECT_4" at 359,298 size 320x40; FormatPattern 999999.999
      ProcessValue <- "WP231PR_DB_DR17_ANA_OUT_VALUE"
      Visibility <- "WP231PR_DB_DR07_SOURCE_ANA_OUT"
   Button "OBJECT_1" at 360,390 size 80x80; TextOn 'Texte / text'; TextOff 'Texte / text'; PictureOff "Save"
      on Release: SetTag("WP231PR_DB_s_CMD2_i_CMD_CODE", '4017'); SetBit("WP231PR_DB_s_CMD2_bo_CMD_TRIGGER")
   IOField "I/O field_2" at 676,304 size 74x27; FormatPattern ????
      Visibility <- "WP231PR_DB_DR07_SOURCE_ANA_OUT"
      ProcessValue <- "WP231PR_DB_DR03_WEIGHT_UNIT"
   TextField "OBJECT_11" at 75,72 size 281x32; Text 'Bereich / Range for Analogue Output / Plage / Scale name'
   TextField "OBJECT_13" at 93,165 size 266x32; Text 'Startwert (0/4mA) / Start value (0/4mA) / Valeur de départ (0/4mA) / Weight Unit'
   TextField "OBJECT_14" at 74,120 size 276x32; Text 'Quelle für Analogsignal / Source for Analogue Signal / Source pour la sortie ana / Scale name'
   IOField "OBJECT_18" at 360,165 size 320x40; FormatPattern 99999.9999
      ProcessValue <- "WP231PR_DB_DR07_START_VAL_ANA_OUT"
   TextField "OBJECT_2" at 143,215 size 216x32; Text 'Endwert (20mA) / End value (20mA) / Valeur de fin (20mA) / Weight Unit'
   IOField "OBJECT_3" at 359,213 size 320x40; FormatPattern 99999.9999
      ProcessValue <- "WP231PR_DB_DR07_END_VAL_ANA_OUT"
   SymbolicIOField "Symbolisches EA-Feld_1" at 362,118 size 320x40; TextOn '1'; TextOff '0'; TextList "007032_SOURCE_ANALOG_OUTPUT"
      ProcessValue <- "WP231PR_DB_DR07_SOURCE_ANA_OUT"
   SymbolicIOField "Symbolisches EA-Feld_3" at 363,69 size 320x40; TextOn '1'; TextOff '0'; TextList "007030_RANGE_ANALOG_OUTPUT"
      ProcessValue <- "WP231PR_DB_DR07_RANGE_ANA_OUT"
   IOField "I/O field_1" at 676,173 size 74x27; FormatPattern ????
      ProcessValue <- "WP231PR_DB_DR03_WEIGHT_UNIT"
   IOField "I/O field_3" at 676,219 size 74x27; FormatPattern ????
      ProcessValue <- "WP231PR_DB_DR03_WEIGHT_UNIT"
   Button "Schaltfläche_1" at 670,390 size 80x80; TextOn 'Texte'; TextOff 'Texte'; PictureOff "Q_Mark"
      on Press: SetBit("S1_SHOW_HELP")
   Softkey "[!Invalid!]Softkey_F6" at -140,-147 size 0x0
      on KeyDown: ActivateScreen("1.5.0.1_Menu_communication_interfaces_1", 0)
   TextField "Textfeld_1" at 0,57 size 800x422; Text 'Um den analogen Ausgang direkt zu Steuern, muss ihm als Quelle "Test / Steuern Ausgang" zugewiesen werden! To test or force the analogue output, the source of the output needs to be set to "Test / Force Output". Pour contrôler directement, à partir du pupitre, la sortie analogique il faut choisir comme source dans le menu 1.5.1 la valeur "Test / Contrôle de la sortie analogique"'
      Visibility <- "S1_SHOW_HELP"
   Button "Schaltfläche_2" at 643,423 size 150x50; TextOn 'Texte'; TextOff 'OK'
      on Press: ResetBit("S1_SHOW_HELP")
      Visibility <- "S1_SHOW_HELP"

screen "1.3.1_DR6_ Limit_values" 800x480, template "Template_1"
   Softkey "[!Invalid!]Softkey_F6" at -140,-147 size 0x0
      on KeyDown: ActivateScreen("Menu_weighing_expert", 0)
   Softkey "[!Invalid!]Softkey_F5" at -140,-147 size 0x0
      on KeyDown: SetTag("S1_CMD2.i_CMD_CODE", 4006); SetTag("S1_CMD2.i_CMD_TRIGGER", 1)
   TextField "Textfeld_3" at 0,58 size 800x422; Text 'Die Ein- und Ausschaltpunkte können für jeden Grenzwert als %-Wert vom Messbereich separat vorgegeben werden. Auf diese Weise kann sowohl eine Minimalwert- und Maximalwertüberwachung mit Hysterese realisiert werden. Zusätzlich kann eine Verzögerungszeit für das Einschalten und Ausschalten vorgegeben werden. Maximalwertüberwachung: ● Einschaltwert > Ausschaltwert Minimalwertüberwachung: ● Einschaltwert < Ausschaltwert The switch-on and switch-off points can be specified separately for each limit value as a percentage of the measuring range. This allows both minimum and maximum value violation monitoring with hysteresis. A delay time for switch-on and switch-off can be specified too. Maximum value monitoring: ● Switch-on value > switch-off value Minimum value monitoring: ● Switch-on value < switch-off value Les valeurs d'enclenchement sont à entrer en % de la plage de mesure'
      Visibility <- "S1_SHOW_HELP"
   Button "Schaltfläche_2" at 643,423 size 150x50; TextOn 'Texte'; TextOff 'OK'
      on Press: ResetBit("S1_SHOW_HELP")
      Visibility <- "S1_SHOW_HELP"
   SymbolicIOField "Symbolisches EA-Feld_1" at 308,331 size 479x34; TextOn '1'; TextOff '0'; TextList "006008_BASIS_FOR_LIMITS_1_2"
      ProcessValue <- "WP231PR_DB_DR06_LIM_REFERENCE"
      Visibility <- "S1_SHOW_HELP"
   TextField "OBJECT_33" at 0,0 size 246x34; Text '1.3.1 Grenzwerte / 1.3.1 Limits / 1.3.1 Limites / Setup 2/3'
   Button "OBJECT_24" at 45,390 size 80x80; TextOn 'Texte / text'; TextOff 'Texte / text'; PictureOff "Exit"
      on Release: ActivateScreen("1.0_Menu_setup", 0)
   TextField "OBJECT_10" at 9,119 size 135x27; Text 'Einschaltwert / Threshold "ON" / Poids enclench. / Display Resolution'
   TextField "OBJECT_12" at 26,169 size 114x27; Text 'Verzögerung / Delay "ON" / Tempo. arrêt / Max. Weight'
   IOField "OBJECT_35" at 375,107 size 130x40; FormatPattern 999.99
      ProcessValue <- "WP231PR_DB_DR06_LIM_2_ON"
   IOField "OBJECT_36" at 375,156 size 130x40; FormatPattern 9999999
      ProcessValue <- "WP231PR_DB_DR06_DELAY_LIM_2_ON"
   IOField "OBJECT_37" at 375,226 size 130x40; FormatPattern 999.99
      ProcessValue <- "WP231PR_DB_DR06_LIM_2_OFF"
   IOField "OBJECT_46" at 375,274 size 130x40; FormatPattern 9999999
      ProcessValue <- "WP231PR_DB_DR06_DELAY_LIM_2_OFF"
   TextField "OBJECT_6" at 3,232 size 142x27; Text 'Ausschaltwert / Threshold "OFF" / Poids arrêt / Calibration Weight'
   TextField "OBJECT_2" at 151,61 size 144x29; Text 'Grenzwert 1 / Limit 1 / Limite 1 / Display Resolution'
   TextField "OBJECT_3" at 380,61 size 144x29; Text 'Grenzwert 2 / Limit 2 / Limite 2 / Display Resolution'
   IOField "OBJECT_4" at 150,107 size 130x40; FormatPattern 999.99
      ProcessValue <- "WP231PR_DB_DR06_LIM_1_ON"
   IOField "OBJECT_5" at 150,156 size 130x40; FormatPattern 9999999
      ProcessValue <- "WP231PR_DB_DR06_DELAY_LIM_1_ON"
   IOField "OBJECT_7" at 150,226 size 130x40; FormatPattern 999.99
      ProcessValue <- "WP231PR_DB_DR06_LIM_1_OFF"
   IOField "OBJECT_8" at 150,274 size 130x40; FormatPattern 9999999
      ProcessValue <- "WP231PR_DB_DR06_DELAY_LIM_1_OFF"
   TextField "OBJECT_9" at 592,61 size 148x29; Text 'Leerbereich / Empty range / Plage vide / Calibration Weight'
   IOField "OBJECT_13" at 591,107 size 130x40; FormatPattern 999.99
      ProcessValue <- "WP231PR_DB_DR06_LIMIT_3_EMPTY"
   IOField "OBJECT_15" at 591,156 size 130x40; FormatPattern 9999999
      ProcessValue <- "WP231PR_DB_DR06_DELAY_EMPTY"
   TextField "OBJECT_11" at 7,276 size 137x27; Text 'Verzögerung / Delay "OFF" / Tempo. marche / Max. Weight'
   TextField "OBJECT_16" at 287,163 size 12x27; Text 's / Calibration Weight'
   TextField "OBJECT_18" at 286,279 size 12x27; Text 's / Calibration Weight'
   TextField "OBJECT_20" at 283,114 size 23x27; Text '% / Calibration Weight'
      Visibility <- "WP231PR_DB_DR06_LIM_REFERENCE"
   TextField "OBJECT_17" at 511,162 size 12x27; Text 's / Calibration Weight'
   TextField "OBJECT_19" at 512,277 size 12x27; Text 's / Calibration Weight'
   Button "OBJECT_1" at 360,390 size 80x80; TextOn 'Texte / text'; TextOff 'Texte / text'; PictureOff "Save"
      on Release: SetTag("WP231PR_DB_s_CMD2_i_CMD_CODE", '4006'); SetBit("WP231PR_DB_s_CMD2_bo_CMD_TRIGGER")
   TextField "OBJECT_27" at 448,360 size 0x34; Text '% / Calibration Weight'
   TextField "OBJECT_28" at 23,335 size 285x27; Text 'Grenzwerte beziehen sich auf: / Limits are related to / Les valeurs limites se réfèrent au: / Display Resolution'
   TextField "OBJECT_30" at 726,161 size 12x27; Text 's / Calibration Weight'
   Button "Schaltfläche_1" at 670,390 size 80x80; TextOn 'Texte'; TextOff 'Texte'; PictureOff "Q_Mark"
      on Press: SetBit("S1_SHOW_HELP")
   IOField "OBJECT_14" at 626,289 size 94x25; FormatPattern 9999999.9
      Visibility <- "WP231PR_DB_DR06_LIM_REFERENCE"
      ProcessValue <- "WP231PR_DB_DR03_MAX_WEIGHT"
   IOField "I/O field_2" at 695,288 size 74x27; FormatPattern ????
      Visibility <- "WP231PR_DB_DR06_LIM_REFERENCE"
      ProcessValue <- "WP231PR_DB_DR03_WEIGHT_UNIT"
   TextField "Textfeld_2" at 593,262 size 160x27; Text 'Max. Wägebereich / Max. weight / poids max'
      Visibility <- "WP231PR_DB_DR06_LIM_REFERENCE"
   IOField "I/O field_1" at 259,113 size 74x27; FormatPattern ????
      Visibility <- "WP231PR_DB_DR06_LIM_REFERENCE"
      ProcessValue <- "WP231PR_DB_DR03_WEIGHT_UNIT"
   IOField "I/O field_3" at 259,232 size 74x27; FormatPattern ????
      Visibility <- "WP231PR_DB_DR06_LIM_REFERENCE"
      ProcessValue <- "WP231PR_DB_DR03_WEIGHT_UNIT"
   TextField "OBJECT_23" at 283,233 size 23x27; Text '% / Calibration Weight'
      Visibility <- "WP231PR_DB_DR06_LIM_REFERENCE"
   TextField "OBJECT_21" at 507,114 size 23x27; Text '% / Calibration Weight'
      Visibility <- "WP231PR_DB_DR06_LIM_REFERENCE"
   TextField "OBJECT_22" at 507,232 size 23x27; Text '% / Calibration Weight'
      Visibility <- "WP231PR_DB_DR06_LIM_REFERENCE"
   TextField "OBJECT_25" at 722,113 size 23x27; Text '% / Calibration Weight'
      Visibility <- "WP231PR_DB_DR06_LIM_REFERENCE"
   IOField "I/O field_4" at 483,113 size 74x27; FormatPattern ????
      Visibility <- "WP231PR_DB_DR06_LIM_REFERENCE"
      ProcessValue <- "WP231PR_DB_DR03_WEIGHT_UNIT"
   IOField "I/O field_5" at 483,232 size 74x27; FormatPattern ????
      Visibility <- "WP231PR_DB_DR06_LIM_REFERENCE"
      ProcessValue <- "WP231PR_DB_DR03_WEIGHT_UNIT"
   IOField "I/O field_6" at 699,113 size 74x27; FormatPattern ????
      Visibility <- "WP231PR_DB_DR06_LIM_REFERENCE"
      ProcessValue <- "WP231PR_DB_DR03_WEIGHT_UNIT"

screen "2.2.1_Scale_Status_1" 800x480, template "Template_1"
   TextField "OBJECT_33" at 0,0 size 387x34; Text '2.2.1 Waagenstatus 1 von 4 / 2.2.1 Scale Status 1 of 4 / 2.2.1 Etat de la balance 1/4 / Setup 1/3'
   Button "OBJECT_24" at 45,390 size 80x80; TextOn 'Texte / text'; TextOff 'Texte / text'; PictureOff "Exit"
      on Release: SetTag("WP231PR_DB_CMD_B", 0)
      on Press: ActivateScreen("2.0_Menu_diagnostic", 0)
   GraphicIOField "OBJECT_304" at 10,233 size 40x30; PictureList "Signal_grey_green"
      ProcessValue <- "WP231PR_DB_s_IO_DATA_SCALE_STATUS_1_STANDSTILL"
   GraphicIOField "OBJECT_305" at 10,91 size 40x30; PictureList "Signal_grey_green"
      ProcessValue <- "WP231PR_DB_s_IO_DATA_SCALE_STATUS_1_D_ZERO"
   GraphicIOField "OBJECT_6" at 10,199 size 40x30; PictureList "Signal_grey_green"
      ProcessValue <- "WP231PR_DB_s_IO_DATA_SCALE_STATUS_1_PRESET_TARE"
   GraphicIOField "OBJECT_12" at 10,127 size 40x30; PictureList "Signal_grey_red"
      ProcessValue <- "WP231PR_DB_s_IO_DATA_SCALE_STATUS_1_MAX_9E"
   TextField "OBJECT_16" at 55,200 size 109x26; Text 'Preset Tara / Preset tare / taré (prédét.) / Error occurred'
   TextField "OBJECT_7" at 236,91 size 54x26; Text 'Leer / Empty / vide / Error occurred'
   TextField "OBJECT_8" at 54,91 size 86x26; Text '1/4d 0 / 1/4d Zero / 1/4 d zéro / Error occurred'
   TextField "OBJECT_9" at 56,236 size 87x26; Text 'Stillstand / Standstill / Etat stable / Error occurred'
   TextField "OBJECT_13" at 55,129 size 85x26; Text '+ Max. 9e / +Max. 9e / +max. 9e / Error occurred'
   GraphicIOField "OBJECT_2" at 10,163 size 40x30; PictureList "Signal_grey_green"
      ProcessValue <- "WP231PR_DB_s_IO_DATA_SCALE_STATUS_1_TARE"
   TextField "OBJECT_3" at 55,164 size 55x26; Text 'Tariert / Tare / taré / Error occurred'
   GraphicIOField "OBJECT_4" at 191,91 size 40x30; PictureList "Signal_grey_yellow"
      ProcessValue <- "WP231PR_DB_s_IO_DATA_SCALE_STATUS_1_EMPTY"
   GraphicIOField "OBJECT_5" at 191,127 size 40x30; PictureList "Signal_grey_yellow"
      ProcessValue <- "WP231PR_DB_s_IO_DATA_SCALE_STATUS_1_LIMIT_1"
   TextField "OBJECT_10" at 236,129 size 99x26; Text 'Grenzwert 1 / Limit 1 / Limite 1 / Error occurred'
   TextField "OBJECT_11" at 236,164 size 99x26; Text 'Grenzwert 2 / Limit 2 / Limite 2 / Error occurred'
   GraphicIOField "OBJECT_31" at 191,163 size 40x30; PictureList "Signal_grey_yellow"
      ProcessValue <- "WP231PR_DB_s_IO_DATA_SCALE_STATUS_1_LIMIT_2"
   TextField "OBJECT_32" at 236,200 size 57x26; Text '< Min. / < min. / Error occurred'
   IOField "OBJECT_301" at 0,40 size 800x40; FormatPattern ????????????????
      ProcessValue <- "WP231PR_DB_DR34_ASCII_DISPLAY"
   TextField "OBJECT_22" at 56,271 size 168x26; Text 'Warten auf Stillstand / Waiting for standstill / Attendre etat stable / Error occurred'
   GraphicIOField "OBJECT_34" at 191,199 size 40x30; PictureList "Signal_grey_yellow"
      ProcessValue <- "WP231PR_DB_s_IO_DATA_SCALE_STATUS_1_BELOW_MIN_WEIGHT"
   GraphicIOField "OBJECT_40" at 10,269 size 40x30; PictureList "Signal_grey_yellow"
      ProcessValue <- "WP231PR_DB_s_IO_DATA_SCALE_STATUS_1_WAITING_FOR_STANDSTILL"
   GraphicIOField "OBJECT_41" at 568,91 size 40x30; PictureList "Signal_grey_green"
      ProcessValue <- "WP231PR_DB_s_IO_DATA_SCALE_STATUS_2_CALIBRATED"
   GraphicIOField "OBJECT_42" at 568,127 size 40x30; PictureList "Signal_grey_yellow"
      ProcessValue <- "WP231PR_DB_s_IO_DATA_SCALE_STATUS_2_SERVICE_MODE"
   GraphicIOField "OBJECT_43" at 568,307 size 40x30; PictureList "Signal_grey_red"
      ProcessValue <- "WP231PR_DB_s_IO_DATA_SCALE_STATUS_2_ERROR"
   GraphicIOField "OBJECT_45" at 568,163 size 40x30; PictureList "Signal_grey_yellow"
      ProcessValue <- "WP231PR_DB_s_IO_DATA_SCALE_STATUS_2_SIMULATION_MODE"
   GraphicIOField "OBJECT_46" at 568,199 size 40x30; PictureList "Signal_grey_green"
      ProcessValue <- "WP231PR_DB_s_IO_DATA_SCALE_STATUS_2_WRITE_PROTECTION"
   GraphicIOField "OBJECT_47" at 568,235 size 40x30; PictureList "Signal_grey_red"
      ProcessValue <- "WP231PR_DB_s_IO_DATA_SCALE_STATUS_2_ANALOGUE_OUT_ERROR"
   GraphicIOField "OBJECT_48" at 568,271 size 40x30; PictureList "Signal_grey_yellow"
      ProcessValue <- "WP231PR_DB_s_IO_DATA_SCALE_STATUS_2_START_UP"
   TextField "OBJECT_51" at 617,273 size 89x26; Text 'Anlauf / Start Up / Démarrage / Error occurred'
   TextField "OBJECT_52" at 615,129 size 113x26; Text 'Servicebetrieb / Service mode / Service / Error occurred'
   TextField "OBJECT_53" at 616,164 size 147x26; Text 'Simulationsmodus / Simulation mode / Mode simulation / Error occurred'
   TextField "OBJECT_54" at 615,91 size 82x26; Text 'Justiert / Calibrated / Etalonnée / Error occurred'
   TextField "OBJECT_55" at 618,202 size 130x26; Text 'P-PR / Write protection / Error occurred'
   TextField "OBJECT_56" at 617,237 size 177x26; Text 'Fehler Analogausgang / Error analogue out / Erreur sortie ana / Error occurred'
   GraphicIOField "OBJECT_18" at 382,127 size 40x30; PictureList "Signal_grey_yellow"
      ProcessValue <- "WP231PR_DB_s_IO_DATA_SCALE_STATUS_2_TRACE"
   GraphicIOField "OBJECT_20" at 382,163 size 40x30; PictureList "Signal_grey_red"
      ProcessValue <- "WP231PR_DB_s_IO_DATA_SCALE_STATUS_2_DIGITAL_INPUT_ERROR"
   GraphicIOField "OBJECT_27" at 382,91 size 40x30; PictureList "Signal_grey_red"
      ProcessValue <- "WP231PR_DB_s_IO_DATA_SCALE_STATUS_2_TIME_BUFFER_ERROR"
   TextField "OBJECT_57" at 429,128 size 98x26; Text 'Trace aktiv / Trace active / Error occurred'
   TextField "OBJECT_58" at 430,165 size 108x26; Text 'Fehler DI / Error DI / Erreur E TOR / Error occurred'
   TextField "OBJECT_62" at 430,94 size 118x26; Text 'Fehler Uhr / Error clock / Erreur Horloge / Error occurred'
   TextField "OBJECT_26" at 616,307 size 66x26; Text 'Störung / Error / Erreur / Error occurred'
   Button "OBJECT_28" at 670,390 size 80x80; TextOn 'Texte / text'; TextOff 'Texte / text'; PictureOff "Right"
      on Release: SetTag("WP231PR_DB_s_CMD2_i_CMD_CODE", '2005'); SetBit("WP231PR_DB_s_CMD2_bo_CMD_TRIGGER")
      on Press: ActivateScreen("2.2.2_Scale_Status_2_DR5", 0)
   Button "Up_to Setup_5_Min_2" at 360,390 size 80x80; TextOn 'Texte / text'; TextOff 'Texte / text'; PictureOff "Home_3"
      on Release: ActivateScreen("0.0.0_Scale_View_1", 0); SetTag("WP231PR_DB_CMD_B", 0)
   Softkey "[!Invalid!]Softkey_F6" at -140,-147 size 0x0
      on KeyDown: function_efd93a16()

screen "2.2.3_Scale_Status_3_DR30" 800x480, template "Template_1"
   TextField "OBJECT_306" at 7,103 size 127x26; Text 'Brutto (Filter 1) / Gross / Brut (Filtre F1) / Scale name'
   IOField "OBJECT_307" at 138,94 size 155x45; FormatPattern 999999.9999
      ProcessValue <- "WP231PR_DB_DR30_GROSS_PROCESS"
   TextField "OBJECT_7" at 7,162 size 121x26; Text 'Netto (Filter 1) / Net / Net (Filtre 1) / Weight Unit'
   IOField "OBJECT_28" at 138,154 size 155x45; FormatPattern 999999.9999
      ProcessValue <- "WP231PR_DB_DR30_NET_PROCESS"
   TextField "OBJECT_8" at 7,218 size 39x26; Text 'Tara / Tare / Depth of Average Value Filter'
   IOField "OBJECT_32" at 138,211 size 155x45; FormatPattern 999999.9999
      ProcessValue <- "WP231PR_DB_DR30_TARE_PROCESS"
   TextField "OBJECT_4" at 7,277 size 127x26; Text 'Brutto (Filter 2) / Gross (F2) / Brut (Filtre F2) / Scale name'
   TextField "OBJECT_5" at 7,333 size 121x26; Text 'Netto (Filter 2) / Net (F2) / Net (Filtre 2) / Weight Unit'
   IOField "OBJECT_6" at 138,266 size 155x45; FormatPattern 999999.9999
      ProcessValue <- "WP231PR_DB_DR30_GROSS_PROCESS_2"
   IOField "OBJECT_10" at 138,324 size 155x45; FormatPattern 999999.9999
      ProcessValue <- "WP231PR_DB_DR30_NET_PROCESS_2"
   TextField "OBJECT_2" at 416,103 size 140x26; Text 'B/N-Gewicht / Gross/Net weight / Poids brut / Net / Scale name'
   TextField "OBJECT_9" at 417,162 size 138x26; Text 'B/N-Gewicht x10 / G/N weight x10 / Brut / Net x 10 / Weight Unit'
   TextField "OBJECT_11" at 417,211 size 141x48; Text 'Tara für Anzeige Tare legal display Tare afficheur certifié Depth of Average Value Filter'
   TextField "OBJECT_12" at 418,270 size 142x48; Text 'Refresh Counter Refresh counter Rafraichissement compteur Scale name'
   IOField "OBJECT_13" at 568,94 size 155x45; FormatPattern 999999.9999
      ProcessValue <- "WP231PR_DB_DR30_GROSS_NET_WEIGHT"
   IOField "OBJECT_14" at 568,154 size 155x45; FormatPattern 999999.9999
      ProcessValue <- "WP231PR_DB_DR30_GROSS_NET_WEIGHT_X10"
   IOField "OBJECT_15" at 567,211 size 155x45; FormatPattern 999999.9999
      ProcessValue <- "WP231PR_DB_DR30_TARE"
   IOField "OBJECT_16" at 567,266 size 155x45; FormatPattern 99999
      ProcessValue <- "WP231PR_DB_DR30_REFRESH_COUNTER"
   TextField "OBJECT_33" at 0,0 size 387x34; Text '2.2.3 Waagenstatus 3 von 4 / 2.2.3 Scale Status 3 of 4 / 2.2.3 Etat de la balance 3/4 / Setup 1/3'
   IOField "I/O field_2" at 293,103 size 74x27; FormatPattern ????
      ProcessValue <- "WP231PR_DB_DR03_WEIGHT_UNIT"
   IOField "I/O field_1" at 293,162 size 74x27; FormatPattern ????
      ProcessValue <- "WP231PR_DB_DR03_WEIGHT_UNIT"
   IOField "I/O field_3" at 293,218 size 74x27; FormatPattern ????
      ProcessValue <- "WP231PR_DB_DR03_WEIGHT_UNIT"
   IOField "I/O field_4" at 293,277 size 74x27; FormatPattern ????
      ProcessValue <- "WP231PR_DB_DR03_WEIGHT_UNIT"
   IOField "I/O field_5" at 293,333 size 74x27; FormatPattern ????
      ProcessValue <- "WP231PR_DB_DR03_WEIGHT_UNIT"
   IOField "I/O field_6" at 723,103 size 74x27; FormatPattern ????
      ProcessValue <- "WP231PR_DB_DR03_WEIGHT_UNIT"
   IOField "I/O field_7" at 723,163 size 74x27; FormatPattern ????
      ProcessValue <- "WP231PR_DB_DR03_WEIGHT_UNIT"
   IOField "I/O field_8" at 723,218 size 74x27; FormatPattern ????
      ProcessValue <- "WP231PR_DB_DR03_WEIGHT_UNIT"
   Button "OBJECT_25" at 545,390 size 80x80; TextOn 'Texte / text'; TextOff 'Texte / text'; PictureOff "Left"
      on Release: ActivateScreen("2.2.2_Scale_Status_2_DR5", 0); SetTag("WP231PR_DB_CMD_B", 2034)
      on Press: SetTag("WP231PR_DB_s_CMD2_i_CMD_CODE", '2005'); SetBit("WP231PR_DB_s_CMD2_bo_CMD_TRIGGER")
   Button "OBJECT_1" at 670,390 size 80x80; TextOn 'Texte / text'; TextOff 'Texte / text'; PictureOff "Right"
      on Release: SetTag("WP231PR_DB_CMD_B", 2031)
      on Press: ActivateScreen("2.2.4_Scale_Status_4_DR31_IO", 0); SetTag("WP231PR_DB_CMD_B", 2031)
   Button "OBJECT_24" at 45,390 size 80x80; TextOn 'Texte / text'; TextOff 'Texte / text'; PictureOff "Exit"
      on Press: ActivateScreen("2.0_Menu_diagnostic", 0); SetTag("WP231PR_DB_CMD_B", 0)
   Button "Up_to Setup_5_Min_2" at 360,390 size 80x80; TextOn 'Texte / text'; TextOff 'Texte / text'; PictureOff "Home_3"
      on Press: ActivateScreen("0.0.0_Scale_View_1", 0); SetTag("WP231PR_DB_CMD_B", 0)
   IOField "OBJECT_301" at 0,40 size 800x40; FormatPattern ????????????????
      ProcessValue <- "WP231PR_DB_DR34_ASCII_DISPLAY"
   Softkey "[!Invalid!]Softkey_F6" at -140,-147 size 0x0
      on KeyDown: ActivateScreen("2.0_Menu_diagnostic", 0)
   Softkey "[!Invalid!]Softkey_F4" at -140,-147 size 0x0
      on KeyDown: ActivateScreen("2.2.4_Scale_Status_4_DR31_IO", 0)

screen "2.2.4_Scale_Status_4_DR31_IO" 800x480, template "Template_1"
   TextField "OBJECT_33" at 0,0 size 387x34; Text '2.2.4 Waagenstatus 4 von 4 / 2.2.4 Scale Status 4 of 4 / 2.2.4 Etat de la balance 4/4 / Setup 1/3'
   TextField "OBJECT_306" at 87,124 size 90x27; Text 'ungefiltert / unfiltered / Non filtré / Scale name'
   IOField "OBJECT_307" at 180,112 size 200x50; FormatPattern 9999999999
      ProcessValue <- "WP231PR_DB_DR31_DIGITS_UNFILTERED"
   IOField "OBJECT_28" at 180,168 size 200x50; FormatPattern 9999999999
      ProcessValue <- "WP231PR_DB_DR31_DIGITS_FILTERED"
   Button "OBJECT_24" at 45,390 size 80x80; TextOn 'Texte / text'; TextOff 'Texte / text'; PictureOff "Exit"
      on Press: ActivateScreen("2.0_Menu_diagnostic", 0); SetTag("WP231PR_DB_CMD_B", 0)
   IOField "OBJECT_32" at 578,112 size 201x50; FormatPattern 9999999999
      ProcessValue <- "WP231PR_DB_DR31_DIGITS_2_FILTERED"
   TextField "OBJECT_3" at 419,124 size 155x27; Text 'gefiltert Filter 2 / Filtered by Filter 2 / Filtré 2 / Scale name'
   TextField "OBJECT_4" at 219,82 size 133x27; Text 'ADC Digitwerte / ADC Digits / Valeur digit CAN / Scale name'
   TextField "OBJECT_5" at 24,180 size 155x27; Text 'gefiltert Filter 1 / Filtered by Filter 1 / Filtré 1 / Scale name'
   TextField "OBJECT_2" at 587,232 size 204x28; Text 'Status Analogausgang / Status Analogue Output / Etat sortie ana / Scale name'
   TextField "OBJECT_6" at 55,236 size 207x28; Text 'Status digitale Eingänge / Status Digital Inputs / Etat entrées TOR / Scale name'
   TextField "OBJECT_7" at 23,291 size 75x27; Text 'DI.0 / Entrée 0 / Scale name'
   TextField "OBJECT_8" at 23,339 size 75x27; Text 'DI.1 / Entrée 1 / Scale name'
   TextField "OBJECT_10" at 145,291 size 75x27; Text 'DI.2 / Entrée 2 / Scale name'
   TextField "OBJECT_11" at 146,339 size 75x27; Text 'DI.3 / Entrée 3 / Scale name'
   TextField "OBJECT_12" at 304,291 size 68x27; Text 'DQ.0 / Sortie 0 / Scale name'
   TextField "OBJECT_13" at 304,339 size 68x27; Text 'DQ.1 / Sortie 1 / Scale name'
   TextField "OBJECT_14" at 432,291 size 68x27; Text 'DQ.2 / Sortie 2 / Scale name'
   TextField "OBJECT_15" at 432,339 size 68x27; Text 'DQ.3 / Sortie 3 / Scale name'
   GraphicIOField "OBJECT_304" at 100,288 size 40x30; PictureList "Signal_grey_yellow"
      ProcessValue <- "WP231PR_DB_DR31_CURRENT_STATE_DI_0"
   GraphicIOField "OBJECT_16" at 100,336 size 38x30; PictureList "Signal_grey_yellow"
      ProcessValue <- "WP231PR_DB_DR31_CURRENT_STATE_DI_1"
   GraphicIOField "OBJECT_17" at 219,288 size 40x30; PictureList "Signal_grey_yellow"
      ProcessValue <- "WP231PR_DB_DR31_CURRENT_STATE_DI_2"
   GraphicIOField "OBJECT_18" at 219,336 size 40x30; PictureList "Signal_grey_yellow"
      ProcessValue <- "WP231PR_DB_DR31_CURRENT_STATE_DI_3"
   GraphicIOField "OBJECT_19" at 372,288 size 40x30; PictureList "Signal_grey_yellow"
      ProcessValue <- "WP231PR_DB_DR31_CURRENT_STATE_DQ_0"
   GraphicIOField "OBJECT_20" at 372,336 size 40x30; PictureList "Signal_grey_yellow"
      ProcessValue <- "WP231PR_DB_DR31_CURRENT_STATE_DQ_1"
   GraphicIOField "OBJECT_21" at 502,288 size 40x30; PictureList "Signal_grey_yellow"
      ProcessValue <- "WP231PR_DB_DR31_CURRENT_STATE_DQ_2"
   GraphicIOField "OBJECT_22" at 502,336 size 40x30; PictureList "Signal_grey_yellow"
      ProcessValue <- "WP231PR_DB_DR31_CURRENT_STATE_DQ_3"
   TextField "OBJECT_1" at 320,234 size 211x28; Text 'Status digitale Ausgänge / Status Digital Outputs / Etat sorties TOR / Scale name'
   Button "OBJECT_25" at 545,390 size 80x80; TextOn 'Texte / text'; TextOff 'Texte / text'; PictureOff "Left"
      on Release: SetTag("WP231PR_DB_CMD_B", 2030)
      on Press: ActivateScreen("2.2.3_Scale_Status_3_DR30", 0)
   Button "Up_to Setup_5_Min_2" at 360,390 size 80x80; TextOn 'Texte / text'; TextOff 'Texte / text'; PictureOff "Home_3"
      on Press: ActivateScreen("0.0.0_Scale_View_1", 0); SetTag("WP231PR_DB_CMD_B", 0)
   IOField "OBJECT_9" at 681,304 size 63x30; FormatPattern 99999
      ProcessValue <- "WP231PR_DB_DR31_CURRENT_ANA_OUT_DIGITS"
   Bar "Balken_1" at 641,271 size 36x106; MinimumValue 0; MaximumValue 65535
      ProcessValue <- "WP231PR_DB_DR31_CURRENT_ANA_OUT_DIGITS"
   TextField "Textfeld_2" at 701,357 size 43x25; Text '0 mA / 0mA'
   TextField "Textfeld_3" at 702,264 size 52x25; Text '24 mA / 24mA'
   TextField "Textfeld_4" at 747,307 size 44x25; Text 'digits'
   IOField "OBJECT_23" at 578,168 size 201x50; FormatPattern 999999999.99
      ProcessValue <- "WP231PR_DB_DR31_LOAD_CELL_SIGNAL"
   TextField "OBJECT_26" at 390,179 size 186x27; Text 'Signalspannung (mV) / load cell signal (mV) / Singal pesons en mV / Scale name'
   IOField "OBJECT_301" at 0,40 size 800x40; FormatPattern ????????????????
      ProcessValue <- "WP231PR_DB_DR34_ASCII_DISPLAY"
   Softkey "[!Invalid!]Softkey_F6" at -140,-147 size 0x0
      on KeyDown: ActivateScreen("2.0_Menu_diagnostic", 0)
   Softkey "[!Invalid!]Softkey_F5" at -140,-147 size 0x0
      on KeyDown: ActivateScreen("2.2.3_Scale_Status_3_DR30", 0)

screen "3.1.1_DR48_Time_language" 800x480, template "Template_1"
   TextField "OBJECT_84" at 0,0 size 439x34; Text '3.1.1 Sprache, Datum & Uhrzeit / 3.1.1 Language, Date & Time / 3.1 Langue, date et heure / Date and time'
   Button "OBJECT_24" at 45,390 size 80x80; TextOn 'Texte / text'; TextOff 'Texte / text'; PictureOff "Exit"
      on Release: function_efd93a16()
   IOField "OBJECT_307" at 248,180 size 90x50; FormatPattern 9999
      ProcessValue <- "WP231PR_DB_DR48_YEAR"
   IOField "OBJECT_1" at 350,180 size 90x50; FormatPattern 99
      ProcessValue <- "WP231PR_DB_DR48_MONTH"
   IOField "OBJECT_3" at 452,180 size 90x50; FormatPattern 99
      ProcessValue <- "WP231PR_DB_DR48_DAY"
   IOField "OBJECT_4" at 248,324 size 90x50; FormatPattern 99
      ProcessValue <- "WP231PR_DB_DR48_HOUR"
   IOField "OBJECT_5" at 350,324 size 90x50; FormatPattern 99
      ProcessValue <- "WP231PR_DB_DR48_MINUTE"
   IOField "OBJECT_6" at 452,324 size 90x50; FormatPattern 99
      ProcessValue <- "WP231PR_DB_DR48_SECOND"
   IOField "OBJECT_7" at 552,324 size 90x50; FormatPattern 999
      ProcessValue <- "WP231PR_DB_DR48_MSECOND"
   Button "OBJECT_8" at 420,390 size 80x80; TextOn 'Texte / text'; TextOff 'Texte / text'; PictureOff "Save"
      on Release: SetTag("WP231PR_DB_s_CMD2_i_CMD_CODE", '2048'); SetBit("WP231PR_DB_s_CMD2_bo_CMD_TRIGGER")
      on Press: SetTag("WP231PR_DB_s_CMD1_i_CMD_CODE", 4048); SetBit("WP231PR_DB_s_CMD1_bo_CMD_TRIGGER")
   TextField "OBJECT_9" at 48,190 size 80x29; Text 'Datum / Date / Error occurred'
   TextField "OBJECT_11" at 48,336 size 80x29; Text 'Zeit / Time / Heure: / Error occurred'
   TextField "Textfeld_1" at 285,300 size 15x25; Text 'H'
   TextField "Textfeld_2" at 386,300 size 17x25; Text 'M'
   TextField "Textfeld_3" at 490,300 size 13x25; Text 'S / s'
   TextField "Textfeld_4" at 582,300 size 26x25; Text 'MS'
   TextField "Textfeld_5" at 284,154 size 16x25; Text 'J / Y / O'
   TextField "Textfeld_6" at 386,154 size 17x25; Text 'M'
   TextField "Textfeld_7" at 489,154 size 16x25; Text 'T / D'
   SymbolicIOField "Symbolisches EA-Feld_1" at 557,187 size 123x34; TextOn '1'; TextOff '0'; TextList "DAY_OF_WEEK"
      ProcessValue <- "WP231PR_DB_DR48_DAY_OF_WEEK"
   GraphicView "Grafikanzeige_4" at 556,84 size 77x54; Picture "Grafik_3"
   Button "OBJECT_96" at 302,80 size 198x60; TextOn 'Texte / text'; TextOff 'Deutsch'
      on Press: function_fb9197e8(L de-DE)
   GraphicView "Grafikanzeige_1" at 304,84 size 70x53; Picture "Grafik_1"
   Button "OBJECT_73" at 46,78 size 200x60; TextOn 'Texte / text'; TextOff 'English'
      on Press: function_fb9197e8(L en-US)
   GraphicView "Grafikanzeige_2" at 49,83 size 66x53; Picture "Grafik_2"
   Softkey "[!Invalid!]Softkey_F6" at -140,-147 size 0x0
      on KeyDown: ActivateScreen("0.0.0_Menu_main", 0)
   Softkey "[!Invalid!]Softkey_F5" at -140,-147 size 0x0
      on KeyDown: SetTag("S1_CMD3.i_CMD_CODE", 4048); SetTag("S1_CMD3.i_CMD_TRIGGER", 1); ActivateScreen("0.0.0_Menu_main", 0)

screen "0.0.0_Menu_main" 800x480, template "Template_1"
   TextField "OBJECT_82" at 0,0 size 205x34; Text 'Hauptmenü / Menu / Menu principal / Main Menu'
   Button "Goto_Service" at 33,73 size 350x90; TextOn 'Texte / text'; TextOff '1.0 Setup / 1.0 Setup / 1.0 Mise en service / Quick Scale Setup'
      on Press: ActivateScreen("1.0_Menu_setup", 0)
   Button "Goto_Diagnostics" at 33,174 size 350x90; TextOn 'Texte / text'; TextOff '2.0 Diagnose / 2.0 Diagnostics / 2.0 Diagnostique / Password'
      on Release: ActivateScreen("2.0_Menu_diagnostic", 0)
   Button "Goto_language_time" at 33,275 size 350x90; TextOn 'Texte / text'; TextOff '3.0 Sprache, Datum & Uhrzeit 3.0 Language, Date & Time 3.0 Langue, date et heure Date and time'
      on Release: ActivateScreen("3.1.1_DR48_Time_language", 0)
      on Press: SetTag("WP231PR_DB_s_CMD2_i_CMD_CODE", 2048); SetBit("WP231PR_DB_s_CMD2_bo_CMD_TRIGGER")
   Button "Exit_to_previous" at 45,390 size 80x80; TextOn 'Texte / text'; TextOff 'Texte / text'; PictureOff "Exit"
      on Press: ActivateScreen("0.0.0_Scale_View_1", 0)
   Softkey "[!Invalid!]Softkey_F6" at -140,-147 size 0x0
      on KeyDown: ActivateScreen("0.0.0_Scale_View_1", 0)

screen "2.4.1_DR9_Modul_info" 800x480, template "Template_1"
   TextField "OBJECT_2" at 0,0 size 260x34; Text '2.4.1 Modul Info / 2.4.1 Modul Info / 2.4.1 Infos module / SIWAREX CSd Module Info'
   TextField "OBJECT_302" at 39,89 size 233x32; Text 'Bestellnummer / Order number / Numéro de commande / Order Number'
   TextField "OBJECT_303" at 41,201 size 85x32; Text 'Version / Version HW'
   TextField "OBJECT_304" at 44,300 size 222x32; Text 'Support Telefon / Support Hotline / Support téléphonique / Version FW'
   IOField "OBJECT_306" at 320,80 size 288x46; FormatPattern ????????????????
      ProcessValue <- "WP231PR_DB_DR09_ORDER_NO"
   IOField "OBJECT_307" at 374,194 size 62x45; FormatPattern 999
      ProcessValue <- "WP231PR_DB_DR09_HARDWARE_VERSION"
   IOField "OBJECT_308" at 570,194 size 60x45; FormatPattern 99
      ProcessValue <- "WP231PR_DB_DR09_FIRMWARE_VERS_POS_1"
   Button "OBJECT_24" at 45,390 size 80x80; TextOn 'Texte / text'; TextOff 'Texte / text'; PictureOff "Exit"
      on Release: ActivateScreen("2.0_Menu_diagnostic", 0)
   IOField "OBJECT_3" at 498,194 size 60x45; FormatPattern ??
      ProcessValue <- "WP231PR_DB_DR09_FIRMWARE_VERS"
   IOField "OBJECT_4" at 648,194 size 60x45; FormatPattern 99
      ProcessValue <- "WP231PR_DB_DR09_FIRMWARE_VERS_POS_2"
   IOField "OBJECT_5" at 725,194 size 60x45; FormatPattern 99
      ProcessValue <- "WP231PR_DB_DR09_FIRMWARE_VERS_POS_3"
   TextField "OBJECT_7" at 41,143 size 169x32; Text 'Seriennummer / Serial number / Numéro de série / Order Number'
   IOField "OBJECT_8" at 320,136 size 290x46; FormatPattern ????????????
      ProcessValue <- "WP231PR_DB_DR09_SERIAL_NO"
   TextField "OBJECT_1" at 42,253 size 213x32; Text 'Version HMI-Projekt / Version HMI-project / Version projet IHM / Version FW'
   TextField "OBJECT_6" at 322,252 size 78x32; Text 'V 2.1.0 / Version FW'
   TextField "OBJECT_9" at 445,200 size 44x32; Text 'FW / Version HW'
   TextField "OBJECT_10" at 320,201 size 48x32; Text 'HW / Version HW'
   TextField "OBJECT_11" at 308,334 size 395x46; Text 'hotline.siwarex@siemens.com / Version FW'
   TextField "OBJECT_12" at 44,341 size 160x32; Text 'Support E-mail / Support e-mail / Version FW'
   TextField "OBJECT_13" at 308,297 size 198x32; Text '+49 721 595 2811 / Version FW'
   Softkey "[!Invalid!]Softkey_F6" at -140,-147 size 0x0
      on KeyDown: ActivateScreen("2.0_Menu_diagnostic", 0)

screen "0.0.0_DR15_Preset_Tare" 800x480, template "Template_1"
   TextField "OBJECT_33" at 0,0 size 196x34; Text 'Taravorgabe / Preset Tare / Consigne Tare / Setup 1/3'
   Button "To_scale_view" at 45,390 size 80x80; TextOn 'Texte / text'; TextOff 'Texte / text'; PictureOff "Exit"
      on Release: function_efd93a16(); SetTag("WP231PR_DB_CMD_B", '0')
      on Press: SetTag("WP231PR_DB_s_CMD2_i_CMD_CODE", 861); SetBit("WP231PR_DB_s_CMD2_bo_CMD_TRIGGER")
   TextField "OBJECT_11" at 155,101 size 167x32; Text 'Taravorgabe 1 / Preset Tare 1 / Tare manuelle 1 / Min. Weight'
   IOField "OBJECT_36" at 320,91 size 200x50; FormatPattern 999999.9999
      ProcessValue <- "WP231PR_DB_DR15_PRESET_TARE_1"
   IOField "EA-Feld_1" at 523,101 size 90x32; FormatPattern ????
      ProcessValue <- "WP231PR_DB_DR03_WEIGHT_UNIT"
   TextField "OBJECT_2" at 152,165 size 167x32; Text 'Taravorgabe 2 / Preset Tare 2 / Tare manuelle 2 / Min. Weight'
   IOField "OBJECT_3" at 320,155 size 200x50; FormatPattern 999999.9999
      ProcessValue <- "WP231PR_DB_DR15_PRESET_TARE_2"
   TextField "OBJECT_4" at 153,229 size 167x32; Text 'Taravorgabe 3 / Preset Tare 3 / Tare manuelle 3 / Min. Weight'
   IOField "OBJECT_5" at 320,219 size 200x50; FormatPattern 999999.9999
      ProcessValue <- "WP231PR_DB_DR15_PRESET_TARE_3"
   Button "T2" at 296,390 size 80x80; TextOn 'Texte / text'; TextOff 'T2 / Menu'; PictureOff "Tare 2"
      on Release: SetTag("WP231PR_DB_s_CMD2_i_CMD_CODE", 2005); SetBit("WP231PR_DB_s_CMD2_bo_CMD_TRIGGER")
      on Press: SetTag("WP231PR_DB_s_CMD1_i_CMD_CODE", 1014); SetBit("WP231PR_DB_s_CMD1_bo_CMD_TRIGGER")
   Button "T1" at 170,390 size 80x80; TextOn 'Texte / text'; TextOff 'T1 / Menu'; PictureOff "Tare 1"
      on Release: SetTag("WP231PR_DB_s_CMD1_i_CMD_CODE", 2005); SetBit("WP231PR_DB_s_CMD1_bo_CMD_TRIGGER")
      on Press: SetTag("WP231PR_DB_s_CMD2_i_CMD_CODE", 1013); SetBit("WP231PR_DB_s_CMD2_bo_CMD_TRIGGER")
   Button "T3" at 420,390 size 80x80; TextOn 'Texte / text'; TextOff 'T3 / Menu'; PictureOff "Tare 3"
      on Release: SetTag("WP231PR_DB_s_CMD2_i_CMD_CODE", 2005); SetBit("WP231PR_DB_s_CMD2_bo_CMD_TRIGGER")
      on Press: SetTag("WP231PR_DB_s_CMD1_i_CMD_CODE", 1015); SetBit("WP231PR_DB_s_CMD1_bo_CMD_TRIGGER")
   TextField "OBJECT_6" at 186,279 size 478x26; Text 'Nach Speichern Tara 1 oder 2 oder 3 aktivieren / After confirmation activate preset tare 1, 2 or 3 / Après confirmation activer tare 1, 2 ou 3 / Min. Weight'
   Button "OBJECT_1" at 545,390 size 80x80; TextOn 'Texte / text'; TextOff 'Texte / text'; PictureOff "Save"
      on Press: SetTag("WP231PR_DB_s_CMD2_i_CMD_CODE", 4015); SetBit("WP231PR_DB_s_CMD2_bo_CMD_TRIGGER")
   TextField "OBJECT_7" at 68,325 size 217x32; Text 'Aktuelle Taravorgabe / current Tare value / Tare actuelle / Min. Weight'
   IOField "OBJECT_15" at 320,316 size 200x50; FormatPattern 99999.9999
      ProcessValue <- "WP231PR_DB_DR05_TARE_WEIGHT_PRESET"
   Button "Schaltfläche_1" at 670,390 size 80x80; TextOn 'Texte'; TextOff 'Texte'; PictureOff "Q_Mark"
      on Press: SetBit("S1_SHOW_HELP")
   IOField "EA-Feld_2" at 523,165 size 90x32; FormatPattern ????
      ProcessValue <- "WP231PR_DB_DR03_WEIGHT_UNIT"
   IOField "EA-Feld_3" at 523,229 size 90x32; FormatPattern ????
      ProcessValue <- "WP231PR_DB_DR03_WEIGHT_UNIT"
   IOField "EA-Feld_4" at 523,325 size 90x32; FormatPattern ????
      ProcessValue <- "WP231PR_DB_DR03_WEIGHT_UNIT"
   IOField "OBJECT_301" at 0,40 size 800x40; FormatPattern ????????????????
      ProcessValue <- "WP231PR_DB_DR34_ASCII_DISPLAY"
   Softkey "[!Invalid!]Softkey_F1" at -140,-147 size 0x0
      on KeyDown: SetTag("S1_CMD3.i_CMD_CODE", 1013); SetTag("S1_CMD3.i_CMD_TRIGGER", 1)
   Softkey "[!Invalid!]Softkey_F2" at -140,-147 size 0x0
      on KeyDown: SetTag("S1_CMD3.i_CMD_CODE", 1014); SetTag("S1_CMD3.i_CMD_TRIGGER", 1)
   Softkey "[!Invalid!]Softkey_F3" at -140,-147 size 0x0
      on KeyDown: SetTag("S1_CMD3.i_CMD_CODE", 1015); SetTag("S1_CMD3.i_CMD_TRIGGER", 1)
   Softkey "[!Invalid!]Softkey_F6" at -140,-147 size 0x0
      on KeyDown: function_efd93a16()
   TextField "Textfeld_1" at 0,57 size 800x422; Text 'Es können bis zu drei Taragewichte vorgegeben werden. Soll ein vordefiniertes Taragewicht zur Anwendung kommen, muss es mit dem entsprechenden Befehl aktiviert werden. Die Taragewichte dürfen den in den erweiterten Waagenparameter festgelegten maximalen Tarawert nicht überschreiten. Beispiel: Nettogewicht = 75,5kg ; Bruttogewicht = 75,5kg ; Taragewicht = 0,0kg Preset Tara 2 = 25,5kg --> Aktivierung Preset-Tara 2 Nettogewicht = 50,0kg ; Bruttogewicht = 75,5kg ; Taragewicht = 25,5kg Up to three predefined tare weights can be entered. If one of them needs to be activated, the corresponding command must be executed. The tare weights may not exceed the maximum tare value defined in the avanced scale parameters. Example: Net Weight = 75,5kg ; Gross Weight = 75,5kg ; Tare Weight = 0,0kg Preset Tare 2 = 25,5kg --> Activation of Preset-Tare 2 Net Weight = 50,0kg ; Gross Weight = 75,5kg ; Tare Weight = 25,5kg 3 valeurs différentes de tare peuvent être entrées'
      Visibility <- "S1_SHOW_HELP"
   Button "Schaltfläche_2" at 643,423 size 150x50; TextOn 'Texte'; TextOff 'OK'
      on Press: ResetBit("S1_SHOW_HELP")
      Visibility <- "S1_SHOW_HELP"

screen "0.0.0_Scale_View_1" 800x480, template "Template_2_Scale_View"
   on GenerateScreen: SetTag("WP231PR_DB_CMD_A", 2034)
   Button "Zero" at 96,390 size 80x80; TextOn 'Texte / text'; TextOff '- 0 - / Menu'; PictureOff "Zero"
      on Release: SetTag("WP231PR_DB_s_CMD2_i_CMD_CODE", 1001); SetBit("WP231PR_DB_s_CMD2_bo_CMD_TRIGGER")
   Button "Tare" at 272,390 size 80x80; TextOn 'Texte / text'; TextOff 'T / Menu'; PictureOff "Tare"
      on Release: SetTag("WP231PR_DB_s_CMD2_i_CMD_CODE", 1011); SetBit("WP231PR_DB_s_CMD2_bo_CMD_TRIGGER")
   Button "Delete_Tare" at 448,390 size 80x80; TextOn 'Texte / text'; TextOff 'TX / Menu'; PictureOff "Del Tare"
      on Release: SetTag("WP231PR_DB_s_CMD2_i_CMD_CODE", 1012); SetBit("WP231PR_DB_s_CMD2_bo_CMD_TRIGGER")
   Button "Goto_preset_tare" at 624,390 size 80x80; TextOn 'Texte / text'; TextOff 'pT / Menu'; PictureOff "pTare"
      on Release: SetTag("WP231PR_DB_CMD_B", 2034); ActivateScreen("0.0.0_DR15_Preset_Tare", 0)
      on Press: SetTag("WP231PR_DB_s_CMD1_i_CMD_CODE", 2015); SetBit("WP231PR_DB_s_CMD1_bo_CMD_TRIGGER")
   Button "Exit_to_Service" at 5,4 size 80x80; TextOn 'Texte / text'; TextOff 'Texte / text'; PictureOff "Menue"
      on Release: ActivateScreen("0.0.0_Menu_main", 0)
   Button "OBJECT_1" at 715,4 size 80x80; TextOn 'Texte / text'; TextOff 'Texte / text'; PictureOff "Diag"
      on Release: ActivateScreen("2.0_Menu_diagnostic", 0)
   Group "Group" at 0,121 size 79x32; Text 'leer'; PictureList "Signal_grey_green"
   Group "Group_2" at 159,121 size 79x32; Text '><'; PictureList "Signal_grey_green"
   Group "Group_3" at 239,121 size 79x32; Text 'T'; PictureList "Signal_grey_green"
   Group "Group_4" at 320,121 size 79x32; Text 'pT'; PictureList "Signal_grey_green"
   Group "Group_5" at 400,121 size 79x32; Text '+9e'; PictureList "Signal_grey_red"
   Group "Group_8" at 640,121 size 84x32; Text 'Service'; PictureList "Signal_grey_yellow"
   IOField "OBJECT_307" at 256,15 size 282x68; FormatPattern ????????????
      ProcessValue <- "WP231PR_DB_DR03_SCALE_NAME"
   Group "Group_6" at 560,121 size 79x32; Text 'GW 2'; PictureList "Signal_grey_yellow"
   Group "Group_7" at 480,121 size 79x32; Text 'GW 1'; PictureList "Signal_grey_yellow"
   Group "Group_9" at 719,121 size 81x32; Text 'Error'; PictureList "Signal_grey_red"
   Group "Group_1" at 80,121 size 79x32; Text '><'; PictureList "Signal_grey_green"
   IOField "OBJECT_301" at 0,167 size 800x160; FormatPattern ????????????????
      ProcessValue <- "WP231PR_DB_DR34_ASCII_DISPLAY"
      Appearance <- "S1_DISPLAY_TAG"
   Button "Button_1" at 0,201 size 800x160; TextOn 'Texte'; TextOff 'Texte'
      on Press: InvertBit("S1_DISPLAY_TAG")
   Softkey "[!Invalid!]Softkey_F5" at -140,-147 size 0x0
      on KeyDown: SetTag("S1_CMD2.i_CMD_CODE", 701); SetTag("S1_CMD2.i_CMD_TRIGGER", 1); ActivateScreen("Scale_View_2", 0)
   Softkey "[!Invalid!]Softkey_F1" at -140,-147 size 0x0
      on KeyDown: SetTag("S1_CMD2.i_CMD_CODE", 1001); SetTag("S1_CMD2.i_CMD_TRIGGER", 1)
   Softkey "[!Invalid!]Softkey_F2" at -140,-147 size 0x0
      on KeyDown: SetTag("S1_CMD3.i_CMD_CODE", 1011); SetTag("S1_CMD3.i_CMD_TRIGGER", 1)
   Softkey "[!Invalid!]Softkey_F3" at -140,-147 size 0x0
      on KeyDown: SetTag("S1_CMD3.i_CMD_CODE", 1012); SetTag("S1_CMD3.i_CMD_TRIGGER", 1)
   Softkey "[!Invalid!]Softkey_F4" at -140,-147 size 0x0
      on KeyDown: SetTag("S1_CMD2.i_CMD_CODE", 2015); SetTag("S1_CMD2.i_CMD_TRIGGER", 1); ActivateScreen("0.0.0_DR15_Preset_Tare", 0)
   Softkey "[!Invalid!]Softkey_F6" at -140,-147 size 0x0
      on KeyDown: ActivateScreen("0.0.0_Menu_main", 0)
   GraphicIOField "OBJECT_304" at 0,121 size 79x32; PictureList "Signal_grey_green"
      ProcessValue <- "WP231PR_DB_s_IO_DATA_SCALE_STATUS_1_EMPTY"
   TextField "OBJECT_7" at 10,124 size 69x27; Text 'leer / empty / vide / Error occurred'
   GraphicIOField "OBJECT_306" at 159,121 size 79x32; PictureList "Signal_grey_green"
      ProcessValue <- "WP231PR_DB_s_IO_DATA_SCALE_STATUS_1_STANDSTILL"
   TextField "OBJECT_21" at 180,124 size 38x27; Text '>< / Error occurred'
   GraphicIOField "OBJECT_3" at 239,121 size 79x32; PictureList "Signal_grey_green"
      ProcessValue <- "WP231PR_DB_s_IO_DATA_SCALE_STATUS_1_TARE"
   TextField "OBJECT_22" at 269,124 size 17x27; Text 'T / Error occurred'
   GraphicIOField "OBJECT_6" at 320,121 size 79x32; PictureList "Signal_grey_green"
      ProcessValue <- "WP231PR_DB_s_IO_DATA_SCALE_STATUS_1_PRESET_TARE"
   TextField "OBJECT_26" at 345,124 size 30x27; Text 'pT / Error occurred'
   GraphicIOField "OBJECT_5" at 400,121 size 79x32; PictureList "Signal_grey_red"
      ProcessValue <- "WP231PR_DB_s_IO_DATA_SCALE_STATUS_1_MAX_9E"
   TextField "OBJECT_27" at 413,124 size 53x27; Text '+9e / +9 e / Error occurred'
   GraphicIOField "OBJECT_4" at 719,121 size 78x32; PictureList "Signal_grey_red"
      ProcessValue <- "WP231PR_DB_s_IO_DATA_SCALE_STATUS_2_ERROR"
   TextField "OBJECT_29" at 732,124 size 68x27; Text 'Error / Erreur / Error occurred'
   GraphicIOField "OBJECT_19" at 640,121 size 79x32; PictureList "Signal_grey_yellow"
      ProcessValue <- "WP231PR_DB_s_IO_DATA_SCALE_STATUS_2_SERVICE_MODE"
   TextField "OBJECT_37" at 644,124 size 80x27; Text 'Service / Error occurred'
   GraphicIOField "OBJECT_45" at 560,121 size 79x32; PictureList "Signal_grey_yellow"
      ProcessValue <- "WP231PR_DB_s_IO_DATA_SCALE_STATUS_1_LIMIT_2"
   TextField "OBJECT_39" at 568,124 size 71x27; Text 'GW 2 / Limit2 / Lim 2 / Error occurred'
   GraphicIOField "OBJECT_44" at 480,121 size 79x32; PictureList "Signal_grey_yellow"
      ProcessValue <- "WP231PR_DB_s_IO_DATA_SCALE_STATUS_1_LIMIT_1"
   TextField "OBJECT_2" at 487,124 size 71x27; Text 'GW 1 / Limit1 / Lim 1 / Error occurred'
   GraphicIOField "OBJECT_8" at 80,121 size 79x32; PictureList "Signal_grey_green"
      ProcessValue <- "WP231PR_DB_s_IO_DATA_SCALE_STATUS_1_D_ZERO"
   TextField "OBJECT_9" at 90,124 size 63x27; Text '1/4d0 / Error occurred'

screen "1.4.1_DR3_Advanced_Scale_Parameters_1" 800x480, template "Template_1"
   TextField "OBJECT_33" at 0,0 size 595x34; Text '1.4.1 Erweiterte Waagenparameter 1 von 5 / 1.4.1 Advanced Scale Parameter 1 of 5 / 1.4.1 Tous les paramètres 1/5 / Setup 1/3'
   Button "Exit_to_service" at 45,390 size 80x80; TextOn 'Texte / text'; TextOff 'Texte / text'; PictureOff "Exit"
      on Release: ActivateScreen("1.0_Menu_setup", 0)
      on Press: SetTag("WP231PR_DB_s_CMD2_i_CMD_CODE", '2'); SetBit("WP231PR_DB_s_CMD2_bo_CMD_TRIGGER")
   Button "OBJECT_1" at 360,390 size 80x80; TextOn 'Texte / text'; TextOff 'Texte / text'; PictureOff "Save"
      on Press: SetTag("WP231PR_DB_s_CMD2_i_CMD_CODE", '4003'); SetBit("WP231PR_DB_s_CMD2_bo_CMD_TRIGGER")
   Button "Exit_to_service_1" at 670,390 size 80x80; TextOn 'Texte / text'; TextOff 'Texte / text'; PictureOff "Right"
      on Press: ActivateScreen("1.4.2_DR3_Advanced_Scale_Parameters_2", 0)
   Group "Group" at 700,5 size 95x30; Text 'Service'; PictureList "Signal_grey_yellow"
   TextField "OBJECT_306" at 230,90 size 179x29; Text 'Waagenname / Scale Name / Nom de la balance / Scale name'
   IOField "OBJECT_307" at 420,84 size 172x40; HelpText 'Name of the Scale (Product, Plant Component or the like). / Nom de la balance'; FormatPattern ????????????
      ProcessValue <- "WP231PR_DB_DR03_SCALE_NAME"
   TextField "OBJECT_7" at 257,141 size 151x29; Text 'Gewichtseinheit / Weight Unit / Unité poids'
   IOField "OBJECT_28" at 420,136 size 172x40; HelpText 'Weight Unit ("g", "kg" or "t" for instance) / Unité poids (par ex. g, kg ou t)'; FormatPattern ????
      ProcessValue <- "WP231PR_DB_DR03_WEIGHT_UNIT"
   TextField "OBJECT_6" at 8,188 size 403x29; Text 'Brutto-Kennung ("B" oder "G") / Indicator for Gross ("B" or "G") / Abréviation pour le poids brut ("B" ou "G") / Weight Unit'
   TextField "OBJECT_9" at 185,285 size 224x29; Text 'Minimaler Wägebereich / Minimum Weight / Poids min / Weight Unit'
   TextField "OBJECT_10" at 156,331 size 254x29; Text 'Maximaler Wägebereich / Maximum Weight / Plage maximale de pesage / Weight Unit'
   TextField "OBJECT_11" at 226,237 size 184x29; Text 'Ziffernschritt (d) / Resolution Step (d) / Résolution (d) / Weight Unit'
   IOField "OBJECT_29" at 420,279 size 172x40; HelpText 'Bei geeichten Waagen mind. 20 x Ziffernschritt d. Bei nicht eichpflichtigen Waagen kann der minimale Wägebereich mit 0 definiert werden. / In legal for trade applications the "Minimum Weight" needs to be at least 20 x resolution step d. In non legal for trade applications the Minimum Weight can be 0. / 20 x d pour usage certifié, sinon pas de limitation (0 par exemple)'; FormatPattern 999
      ProcessValue <- "WP231PR_DB_DR03_MIN_WEIGHT_D"
   IOField "OBJECT_12" at 420,325 size 173x40; HelpText 'Maximales Gewicht auf der Waage. Bei geeichten Waagen bitte entsprechende Einschränkungen berücksichtigen! / Maximum weight applied on the scale. Consider restrictions for legal for trade scales. / Poids max. sur la balance'; FormatPattern 9999999.9999
      ProcessValue <- "WP231PR_DB_DR03_MAX_WEIGHT"
   IOField "OBJECT_13" at 420,230 size 172x40; HelpText 'Resolution of the scale. If the Weight Unit is defined as "kg" a resolution of 0,1 effects a resolution step of 0,1kg. / Résolution de la balance. Avec un unité de poids de 1kg, la résolution de 0,1 signifie 0,1kg'; FormatPattern 9999.9999
      ProcessValue <- "WP231PR_DB_DR03_RESOLUTION_D"
   IOField "I/O field_2" at 596,325 size 60x40; FormatPattern ????
      ProcessValue <- "WP231PR_DB_DR03_WEIGHT_UNIT"
   TextField "Textfeld_1" at 636,284 size 18x29; Text 'x'
   IOField "I/O field_1" at 596,232 size 60x40; FormatPattern ????
      ProcessValue <- "WP231PR_DB_DR03_WEIGHT_UNIT"
   TextField "OBJECT_2" at 605,284 size 16x29; Text 'd / Weight Unit'
   SymbolicIOField "Symbolic I/O field_1" at 421,187 size 172x31; TextOn '1'; TextOff '0'; TextList "003030_LETTER_FOR_GROSS_WEIGHT"
      ProcessValue <- "WP231PR_DB_DR03_LETTER_GROSS_WEIGHT_2"
   Softkey "[!Invalid!]Softkey_F6" at -140,-147 size 0x0
      on KeyDown: ActivateScreen("Menu_weighing_expert", 0)
   Softkey "[!Invalid!]Softkey_F5" at -140,-147 size 0x0
      on KeyDown: SetTag("S1_CMD2.i_CMD_CODE", 4003); SetTag("S1_CMD2.i_CMD_TRIGGER", 1)
   GraphicIOField "OBJECT_19" at 765,5 size 30x30; PictureList "Signal_grey_yellow"
      ProcessValue <- "WP231PR_DB_s_IO_DATA_SCALE_STATUS_2_SERVICE_MODE"
   TextField "OBJECT_37" at 700,7 size 57x25; Text 'Service / Error occurred'
   TextField "Textfeld_2" at 0,57 size 800x422; Text 'Waagenname : Name der Waage (Produkt, Ort, Anlagenteil, o.Ä.) Gewichtseinheit : Frei wählbar - keine direkte Relation zu Ziffernschritt Brutto-Kennung : B für "Brutto" oder G für "Brutto" Ziffernschritt (d) : Einheit "kg" --> 0,1 = 100g - Schritte, 1 = 1kg - Schritte Minimaler Wägebereich : Bei eichfähigen Waagen mindestens 20 x d, ansonsten 0. Maximaler Wägebereich : Bei eichfähigen Waagen 3000 oder 6000 x d, ansonsten maximale Last der Waage. Scale Name : Name of the scale (Product, Location, Plant, or the like) Weight Unit : Free selectable - no direct relation to the resolution Gross Indicator : B for "Gross" or G for "Gross" Resolution (d) : Unit "kg" --> 0,1 = 100g - steps, 1 = 1kg - steps Minimum Weight : Legal for trade --> min. 20 x d, otherwise 0. Maximum Weight : Legal for trade 3000 or 6000 x d, otherwise nominal load of the scale. Nom de la balance: (Produit, lieux d'installation,..'
      Visibility <- "S1_SHOW_HELP"
   Button "Schaltfläche_2" at 643,423 size 150x50; TextOn 'Texte'; TextOff 'OK'
      on Press: ResetBit("S1_SHOW_HELP")
      Visibility <- "S1_SHOW_HELP"

screen "1.2.1_Quick_Start_1" 800x480, template "Template_1"
   TextField "OBJECT_33" at 0,0 size 440x34; Text '1.2.1 Quick Start 1 von 5 / 1.2.1 Quick Start 1 of 5 / 1.2.1 Mise en service rapide 1/5 / Setup 1/3'
   Button "Exit to Service" at 45,390 size 80x80; TextOn 'Texte / text'; TextOff 'Texte / text'; PictureOff "Exit"
      on Release: ActivateScreen("1.0_Menu_setup", 0)
      on Press: SetTag("WP231PR_DB_s_CMD2_i_CMD_CODE", '2'); SetBit("WP231PR_DB_s_CMD2_bo_CMD_TRIGGER")
   Button "Factory settings" at 110,112 size 580x90; TextOn 'Texte / text'; TextOff '"Quick Start" mit bestehenden Einstellungen / Run "Quick Start" with existing settings / Démarrage rapide avec les paramètres actuels / Acknowledge Empty Bin'
      on Release: ActivateScreen("1.2.2_Quick_Start_2", 0)
      on Press: SetTag("WP231PR_DB_s_CMD2_i_CMD_CODE", '2003'); SetBit("WP231PR_DB_s_CMD2_bo_CMD_TRIGGER")
   Group "Group" at 700,5 size 95x30; Text 'Service'; PictureList "Signal_grey_yellow"
   Button "Factory settings_1" at 110,237 size 580x90; TextOn 'Texte / text'; TextOff '"Quick Start" mit Werkseinstellungen / Run "Quick Start" with factory default settings / Démarrage rapide avec les paramètres usine / Acknowledge Empty Bin'
      on Release: ActivateScreen("1.2.2_Quick_Start_2", 0); SetTag("WP231PR_DB_s_CMD2_i_CMD_CODE", '2003'); SetBit("WP231PR_DB_s_CMD2_bo_CMD_TRIGGER")
      on Press: SetTag("WP231PR_DB_s_CMD1_i_CMD_CODE", 12); SetBit("WP231PR_DB_s_CMD1_bo_CMD_TRIGGER")
   Button "Schaltfläche_1" at 360,390 size 80x80; TextOn 'Texte'; TextOff 'Texte'; PictureOff "Q_Mark"
      on Press: SetBit("S1_SHOW_HELP")
   Softkey "[!Invalid!]Softkey_F6" at -140,-147 size 0x0
      on KeyDown: ActivateScreen("1.0_Menu_setup", 0)
   Softkey "[!Invalid!]Softkey_F5" at -140,-147 size 0x0
      on KeyDown: SetTag("S1_CMD2.i_CMD_CODE", 2010); SetTag("S1_CMD2.i_CMD_TRIGGER", 1); SetTag("S1_CMD3.i_CMD_CODE", 2003); SetTag("S1_CMD3.i_CMD_TRIGGER", 1); ActivateScreen("1.2.6_Quick_Start_4", 0)
   GraphicIOField "OBJECT_19" at 765,5 size 30x30; PictureList "Signal_grey_yellow"
      ProcessValue <- "WP231PR_DB_s_IO_DATA_SCALE_STATUS_2_SERVICE_MODE"
   TextField "OBJECT_37" at 700,7 size 57x25; Text 'Service / Error occurred'
   TextField "Textfeld_1" at 0,57 size 800x422; Text '"Quick Start" ermöglicht eine schnelle Basis-Inbetriebnahme der Waage. Es besteht die Möglichkeit die Waage mit oder ohne Justagegewichte zu justieren. "Quick Start" kann mit den bestehenden Waagenparametern, als auch mit geladenen Werkseinstellungen durchgeführt werden. "Quick Start" allows a fast and easy basic commissioning of the scale. It is possible to calibrate the scale with or without calibration weights. You can enter the "Quick Start" procedure with loaded factory settings or with maintaining the scale settings. Le démarrage rapide pour une mise en service en quelques minutes'
      Visibility <- "S1_SHOW_HELP"
   Button "Schaltfläche_2" at 643,423 size 150x50; TextOn 'Texte'; TextOff 'OK'
      on Press: ResetBit("S1_SHOW_HELP")
      Visibility <- "S1_SHOW_HELP"

screen "1.2.6_Quick_Start_4" 800x480, template "Template_1"
   TextField "OBJECT_33" at 0,0 size 662x34; Text '1.2.6 Quick Start 4 von 5 / 1.2.6 Quick Start 4 of 5 - Load Cells Parameters / 1.2.6 Mise en service rapide 4/5 / Setup 1/3'
   Button "Down to Setup_5_Min_03" at 670,390 size 80x80; TextOn 'Texte / text'; TextOff 'Texte / text'; PictureOff "Right"
      on Release: ActivateScreen("1.2.7_Quick_Start_Automatic_Calibration", 0)
      on Press: SetTag("WP231PR_DB_CMD_A", 2034)
   TextField "OBJECT_7" at 297,150 size 264x32; Text 'Anzahl Auflagepunkte / Number of support points / Nombre de points d'appui / Weight Unit'
   IOField "OBJECT_28" at 580,142 size 130x45; HelpText 'Bei Silo mit drei Beinen = 3 Bei Silo mit vier Beinen = 4 usw. Hopper with 3 legs = 3 Hopper with 4 legs = 4 ASO. 3 pour un silo avec 3 pieds, 4 pour un silo à 4 pieds etc.'; FormatPattern 9
      ProcessValue <- "WP231PR_DB_DR10_NO_POINTS_OF_SUPPORT"
   Button "Exit to Service" at 45,390 size 80x80; TextOn 'Texte / text'; TextOff 'Texte / text'; PictureOff "Exit"
      on Press: SetTag("WP231PR_DB_s_CMD2_i_CMD_CODE", '2'); SetBit("WP231PR_DB_s_CMD2_bo_CMD_TRIGGER")
      on Release: ActivateScreen("1.0_Menu_setup", 0)
   TextField "OBJECT_308" at 201,259 size 358x32; Text 'Nennlast einer Wägezelle / Nominal load of one single load cell / Charge nominale d'un peson / Limit Freq. Low Pass Filter'
   TextField "OBJECT_9" at 39,206 size 528x32; Text 'Durchschnittskennwert aller Wägezellen (mV/V) / Average of all characteristic values (mV/V) / Valeur moyenne de la sensibilité des pesons (mV/V) / Stand Still Time'
   IOField "OBJECT_32" at 580,198 size 130x45; HelpText 'Kennwert Zelle 1 = 1,998 mV/V Kennwert Zelle 2 = 2,002 mV/V Kennwert Zelle 3 = 2,000 mV/V ======================== Durchschnitt = 2,000 mV/V Charact. Value Cell 1 = 1,998 mV/V Charact. Value Cell 2 = 2,002 mV/V Charact. Value Cell 3 = 2,000 mV/V =========================== Average = 2,000 mV/V Sensibilité peson 1 = 1,998 mV/V Sensibilité peson 2 = 2,002 mV/V Sensibilité peson 3 = 2,000 mV/V ======================== Moyenne = 2,000 mV/V'; FormatPattern 99.999999
      ProcessValue <- "WP231PR_DB_DR10_GAIN_LOAD_CELL"
   IOField "OBJECT_2" at 580,252 size 130x45; FormatPattern 999999999.9
      ProcessValue <- "WP231PR_DB_DR10_NOM_LOAD_ONE_LOAD_CELL"
   Button "Up_to Setup_5_Min_01" at 545,390 size 80x80; TextOn 'Texte / text'; TextOff 'Texte / text'; PictureOff "Left"
      on Release: ActivateScreen("1.2.3_Quick_Start_3", 0)
   IOField "I/O field_2" at 713,261 size 82x29; FormatPattern ????
      ProcessValue <- "WP231PR_DB_DR03_WEIGHT_UNIT"
   Group "Group" at 700,5 size 95x30; Text 'Service'; PictureList "Signal_grey_yellow"
   Button "Down to Setup_5_Min_1" at 360,390 size 80x80; TextOn 'Texte / text'; TextOff 'Texte / text'; PictureOff "Save"
      on Press: SetTag("WP231PR_DB_s_CMD1_i_CMD_CODE", 4010); SetBit("WP231PR_DB_s_CMD1_bo_CMD_TRIGGER")
   Softkey "[!Invalid!]Softkey_F5" at -140,-147 size 0x0
      on KeyDown: SetTag("S1_CMD3.i_CMD_CODE", 4010); SetTag("S1_CMD3.i_CMD_TRIGGER", 1); SetTag("S1_CMD2.i_CMD_CODE", 4003); SetTag("S1_CMD2.i_CMD_TRIGGER", 1); ActivateScreen("1.2.3_Quick_Start_3", 0)
   Softkey "[!Invalid!]Softkey_F6" at -140,-147 size 0x0
      on KeyDown: ActivateScreen("1.0_Menu_setup", 0)
   Softkey "[!Invalid!]Softkey_F4" at -140,-147 size 0x0
      on KeyDown: ActivateScreen("1.2.1_Quick_Start_1", 0)
   GraphicIOField "OBJECT_19" at 765,5 size 30x30; PictureList "Signal_grey_yellow"
      ProcessValue <- "WP231PR_DB_s_IO_DATA_SCALE_STATUS_2_SERVICE_MODE"
   TextField "OBJECT_37" at 700,7 size 57x25; Text 'Service / Error occurred'

screen "1.2.3_Quick_Start_3" 800x480, template "Template_1"
   TextField "OBJECT_35" at 0,0 size 440x34; Text '1.2.3 Quick Start 3 von 5 / 1.2.3 Quick Start 3 of 5 / 1.2.3 Mise en service rapide 3/5 / Quick Setup'
   Button "Exit to Service" at 45,390 size 80x80; TextOn 'Texte / text'; TextOff 'Texte / text'; PictureOff "Exit"
      on Release: ActivateScreen("1.0_Menu_setup", 0)
      on Press: SetTag("WP231PR_DB_s_CMD2_i_CMD_CODE", '2'); SetBit("WP231PR_DB_s_CMD2_bo_CMD_TRIGGER")
   TextField "OBJECT_38" at 34,80 size 762x32; Text 'Soll die Waage mit oder ohne Gewichte justiert werden? / Do you want to calibrate the scale with or without weights? / Calibration avec ou sans poids étalon? / For Quick Setup the scale must be empty'
   Button "Up_to Setup_5_Min_01" at 545,390 size 80x80; TextOn 'Texte / text'; TextOff 'Texte / text'; PictureOff "Left"
      on Release: ActivateScreen("1.2.2_Quick_Start_2", 0)
   Group "Group" at 700,5 size 95x30; Text 'Service'; PictureList "Signal_grey_yellow"
   Button "Factory settings" at 110,138 size 580x90; TextOn 'Texte / text'; TextOff 'Mit Gewichten justieren / Calibrate With Weights / Etalonner avec des poids étalons / Acknowledge Empty Bin'
      on Release: ActivateScreen("1.2.4_Quick_Start_Manual_Calibration_1", 0)
   Button "Factory settings_1" at 110,263 size 580x90; TextOn 'Texte / text'; TextOff 'Ohne Gewichte justieren (automatisch) Calibrate without weights (automatic) Calibration sans poids étalon Acknowledge Empty Bin'
      on Release: ActivateScreen("1.2.6_Quick_Start_4", 0)
      on Press: SetTag("WP231PR_DB_s_CMD2_i_CMD_CODE", '2010'); SetBit("WP231PR_DB_s_CMD2_bo_CMD_TRIGGER")
   Button "Schaltfläche_1" at 360,390 size 80x80; TextOn 'Texte'; TextOff 'Texte'; PictureOff "Q_Mark"
      on Press: SetBit("S1_SHOW_HELP")
   Softkey "[!Invalid!]Softkey_F6" at -140,-147 size 0x0
      on KeyDown: SetTag("S1_CMD3.i_CMD_CODE", 2); SetTag("S1_CMD3.i_CMD_TRIGGER", 1); ActivateScreen("1.0_Menu_setup", 0)
   Softkey "[!Invalid!]Softkey_F4" at -140,-147 size 0x0
      on KeyDown: ActivateScreen("1.2.6_Quick_Start_4", 0)
   GraphicIOField "OBJECT_19" at 765,5 size 30x30; PictureList "Signal_grey_yellow"
      ProcessValue <- "WP231PR_DB_s_IO_DATA_SCALE_STATUS_2_SERVICE_MODE"
   TextField "OBJECT_37" at 700,7 size 57x25; Text 'Service / Error occurred'
   TextField "Textfeld_1" at 0,57 size 800x422; Text 'Justage mit Gewichten: Es müssen mindestens 5% der Nennlast der Waage als Justagegewicht zur Verfügung stehen. Beispiel: 3 x 2t Wägezellen = 6t Nennlast --> Die Waage muss mit mindestens 300kg (5% von 6t) justiert werden. Wird der Justagepunkt 2 ebenfalls genutzt, muss dieser wiederum mindestens 300kg vom Justagepunkt 1 entfernt sein. Automatische Justage: Es sind keine Justagegewichte notwendig. Die Wägezellendaten müssen zur Verfügung stehen. Mechanische Einflüsse werden nicht berücksichtigt! Calibration with Weights: At least 5% of the nominal load of the scale are neccessary for the calibration. Example: 3 x 2t loadcells = 6t nominal load --> The scale must be calibrated with 300kg (5% of 6t) at least. If calibration point 2 is used too, the difference between calibration point 1 and 2 must be again at least 300kg. Automatic Calibration: No calibration weights are required. The loadcell data must be available. Mechanical influences are not considered! Etalonnage avec un poids étalon. Au min 5% de la charge nominale des pesons'
      Visibility <- "S1_SHOW_HELP"
   Button "Schaltfläche_2" at 643,423 size 150x50; TextOn 'Texte'; TextOff 'OK'
      on Press: ResetBit("S1_SHOW_HELP")
      Visibility <- "S1_SHOW_HELP"

